  MoveL 6660 to (240.24, 47.55, 97.46) mm, rotated rx 180 ry 0 rz 180 deg; joints [-155.614, -72.061, -46.003, 43.936, 36.516, -37.754]
  Call Extruder(209.25610)
  MoveL 6661 to (240.29, 47.8, 97.46) mm, rotated rx 180 ry 0 rz 180 deg; joints [-155.594, -72.082, -45.96, 43.985, 36.511, -37.802]
  MoveL 6662 to (240.29, 47.8, 97.46) mm, rotated rx 180 ry 0 rz 180 deg; joints [-155.594, -72.082, -45.96, 43.985, 36.511, -37.802]
  Call Extruder(209.39246)
  MoveL 6663 to (240.34, 48.05, 97.46) mm, rotated rx -180 ry 0 rz 180 deg; joints [-155.574, -72.103, -45.916, 44.033, 36.507, -37.85]
  MoveL 6664 to (240.34, 48.05, 97.46) mm, rotated rx -180 ry 0 rz 180 deg; joints [-155.574, -72.103, -45.916, 44.033, 36.507, -37.85]
  Call Extruder(209.52822)
  MoveL 6665 to (240.39, 48.3, 97.46) mm, rotated rx -180 ry 0 rz 180 deg; joints [-155.554, -72.123, -45.873, 44.081, 36.503, -37.899]
  MoveL 6666 to (240.39, 48.3, 97.46) mm, rotated rx -180 ry 0 rz 180 deg; joints [-155.554, -72.123, -45.873, 44.081, 36.503, -37.899]
  Call Extruder(209.66337)
  MoveL 6667 to (240.44, 48.55, 97.46) mm, rotated rx 180 ry 0 rz 180 deg; joints [-155.534, -72.144, -45.829, 44.129, 36.499, -37.947]
  MoveL 6668 to (240.44, 48.55, 97.46) mm, rotated rx 180 ry 0 rz 180 deg; joints [-155.534, -72.144, -45.829, 44.129, 36.499, -37.947]
  Call Extruder(209.79791)
  MoveL 6669 to (240.49, 48.8, 97.46) mm, rotated rx 180 ry 0 rz 180 deg; joints [-155.514, -72.165, -45.785, 44.177, 36.495, -37.995]
  MoveL 6670 to (240.49, 48.8, 97.46) mm, rotated rx 180 ry 0 rz 180 deg; joints [-155.514, -72.165, -45.785, 44.177, 36.495, -37.995]
  Call Extruder(209.93183)
  MoveL 6671 to (240.54, 49.05, 97.46) mm, rotated rx 180 ry 0 rz -180 deg; joints [-155.494, -72.186, -45.742, 44.226, 36.491, -38.043]
  MoveL 6672 to (240.54, 49.05, 97.46) mm, rotated rx 180 ry 0 rz -180 deg; joints [-155.494, -72.186, -45.742, 44.226, 36.491, -38.043]
  Call Extruder(210.07970)
  MoveL 6673 to (240.59, 49.33, 97.46) mm, rotated rx 180 ry 0 rz 180 deg; joints [-155.471, -72.208, -45.695, 44.279, 36.487, -38.096]
  MoveL 6674 to (240.59, 49.33, 97.46) mm, rotated rx 180 ry 0 rz 180 deg; joints [-155.471, -72.208, -45.695, 44.279, 36.487, -38.096]
  Call Extruder(210.24144)
  MoveL 6675 to (240.64, 49.63, 97.46) mm, rotated rx 180 ry 0 rz -180 deg; joints [-155.446, -72.232, -45.644, 44.337, 36.484, -38.154]
  MoveL 6676 to (240.64, 49.63, 97.46) mm, rotated rx 180 ry 0 rz -180 deg; joints [-155.446, -72.232, -45.644, 44.337, 36.484, -38.154]
  Call Extruder(210.40246)
  MoveL 6677 to (240.69, 49.94, 97.46) mm, rotated rx 180 ry 0 rz 180 deg; joints [-155.421, -72.256, -45.593, 44.395, 36.481, -38.212]
  MoveL 6678 to (240.69, 49.94, 97.46) mm, rotated rx 180 ry 0 rz 180 deg; joints [-155.421, -72.256, -45.593, 44.395, 36.481, -38.212]
  Call Extruder(210.56275)
  MoveL 6679 to (240.74, 50.24, 97.46) mm, rotated rx -180 ry 0 rz 180 deg; joints [-155.396, -72.28, -45.543, 44.453, 36.477, -38.27]
  MoveL 6680 to (240.74, 50.24, 97.46) mm, rotated rx -180 ry 0 rz 180 deg; joints [-155.396, -72.28, -45.543, 44.453, 36.477, -38.27]
  Call Extruder(210.72231)
  MoveL 6681 to (240.78, 50.55, 97.46) mm, rotated rx 180 ry 0 rz 180 deg; joints [-155.371, -72.305, -45.492, 44.512, 36.474, -38.328]
  MoveL 6682 to (240.78, 50.55, 97.46) mm, rotated rx 180 ry 0 rz 180 deg; joints [-155.371, -72.305, -45.492, 44.512, 36.474, -38.328]
  Call Extruder(210.88114)
  MoveL 6683 to (240.83, 50.86, 97.46) mm, rotated rx -180 ry 0 rz 180 deg; joints [-155.346, -72.329, -45.441, 44.57, 36.47, -38.386]
  MoveL 6684 to (240.83, 50.86, 97.46) mm, rotated rx -180 ry 0 rz 180 deg; joints [-155.346, -72.329, -45.441, 44.57, 36.47, -38.386]
  Call Extruder(211.05982)
  MoveL 6685 to (240.88, 51.2, 97.46) mm, rotated rx -180 ry 0 rz 180 deg; joints [-155.317, -72.355, -45.386, 44.636, 36.467, -38.451]
  MoveL 6686 to (240.88, 51.2, 97.46) mm, rotated rx -180 ry 0 rz 180 deg; joints [-155.317, -72.355, -45.386, 44.636, 36.467, -38.451]
  Call Extruder(211.25826)
  MoveL 6687 to (240.93, 51.59, 97.46) mm, rotated rx 180 ry 0 rz -180 deg; joints [-155.285, -72.384, -45.325, 44.708, 36.465, -38.522]
  MoveL 6688 to (240.93, 51.59, 97.46) mm, rotated rx 180 ry 0 rz -180 deg; joints [-155.285, -72.384, -45.325, 44.708, 36.465, -38.522]
  Call Extruder(211.45583)
  MoveL 6689 to (240.97, 51.98, 97.46) mm, rotated rx 180 ry 0 rz 180 deg; joints [-155.252, -72.413, -45.264, 44.781, 36.463, -38.594]
  MoveL 6690 to (240.97, 51.98, 97.46) mm, rotated rx 180 ry 0 rz 180 deg; joints [-155.252, -72.413, -45.264, 44.781, 36.463, -38.594]
  Call Extruder(211.65254)
  MoveL 6691 to (241.02, 52.36, 97.46) mm, rotated rx 180 ry 0 rz 180 deg; joints [-155.22, -72.442, -45.204, 44.854, 36.46, -38.666]
  MoveL 6692 to (241.02, 52.36, 97.46) mm, rotated rx 180 ry 0 rz 180 deg; joints [-155.22, -72.442, -45.204, 44.854, 36.46, -38.666]
  Call Extruder(211.84838)
  MoveL 6693 to (241.06, 52.75, 97.46) mm, rotated rx 180 ry 0 rz 180 deg; joints [-155.188, -72.471, -45.143, 44.926, 36.458, -38.738]
  MoveL 6694 to (241.06, 52.75, 97.46) mm, rotated rx 180 ry 0 rz 180 deg; joints [-155.188, -72.471, -45.143, 44.926, 36.458, -38.738]
  Call Extruder(212.14382)
  MoveL 6695 to (241.11, 53.34, 97.46) mm, rotated rx 180 ry 0 rz 180 deg; joints [-155.138, -72.512, -45.057, 45.035, 36.457, -38.844]
  MoveL 6696 to (241.11, 53.34, 97.46) mm, rotated rx 180 ry 0 rz 180 deg; joints [-155.138, -72.512, -45.057, 45.035, 36.457, -38.844]
  Call Extruder(212.43792)
  MoveL 6697 to (241.16, 53.93, 97.46) mm, rotated rx 180 ry 0 rz 180 deg; joints [-155.088, -72.553, -44.97, 45.144, 36.457, -38.951]
  MoveL 6698 to (241.16, 53.93, 97.46) mm, rotated rx 180 ry 0 rz 180 deg; joints [-155.088, -72.553, -44.97, 45.144, 36.457, -38.951]
  Call Extruder(212.73070)
  MoveL 6699 to (241.2, 54.52, 97.46) mm, rotated rx 180 ry 0 rz -180 deg; joints [-155.038, -72.595, -44.883, 45.253, 36.456, -39.058]
  MoveL 6700 to (241.2, 54.52, 97.46) mm, rotated rx 180 ry 0 rz -180 deg; joints [-155.038, -72.595, -44.883, 45.253, 36.456, -39.058]
  Call Extruder(213.30415)
  MoveL 6701 to (241.25, 55.68, 97.46) mm, rotated rx 180 ry 0 rz 180 deg; joints [-154.938, -72.671, -44.724, 45.464, 36.461, -39.263]
  MoveL 6702 to (241.25, 55.68, 97.46) mm, rotated rx 180 ry 0 rz 180 deg; joints [-154.938, -72.671, -44.724, 45.464, 36.461, -39.263]
  Call Extruder(214.01798)
  MoveL 6703 to (241.29, 57.14, 97.46) mm, rotated rx 180 ry 0 rz -180 deg; joints [-154.812, -72.765, -44.527, 45.727, 36.469, -39.518]
  Call Extruder(256.08287)
  MoveL 6704 to (241.29, 142.86, 97.46) mm, rotated rx 180 ry 0 rz 180 deg; joints [-147.778, -79.586, -30.484, 61.433, 37.381, -55.581]
  Call Extruder(256.51129)
  MoveL 6705 to (241.27, 143.73, 97.46) mm, rotated rx 180 ry 0 rz 180 deg; joints [-147.711, -79.673, -30.306, 61.599, 37.394, -55.761]
  MoveL 6706 to (241.27, 143.73, 97.46) mm, rotated rx 180 ry 0 rz 180 deg; joints [-147.711, -79.673, -30.306, 61.599, 37.394, -55.761]
  Call Extruder(257.08474)
  MoveL 6707 to (241.22, 144.9, 97.46) mm, rotated rx -180 ry 0 rz -180 deg; joints [-147.62, -79.787, -30.075, 61.818, 37.413, -55.998]
  MoveL 6708 to (241.22, 144.9, 97.46) mm, rotated rx -180 ry 0 rz -180 deg; joints [-147.62, -79.787, -30.075, 61.818, 37.413, -55.998]
  Call Extruder(257.51908)
  MoveL 6709 to (241.18, 145.77, 97.46) mm, rotated rx 180 ry 0 rz 180 deg; joints [-147.551, -79.872, -29.904, 61.981, 37.43, -56.174]
  MoveL 6710 to (241.18, 145.77, 97.46) mm, rotated rx 180 ry 0 rz 180 deg; joints [-147.551, -79.872, -29.904, 61.981, 37.43, -56.174]
  Call Extruder(257.81319)
  MoveL 6711 to (241.13, 146.36, 97.46) mm, rotated rx -180 ry 0 rz -180 deg; joints [-147.504, -79.926, -29.794, 62.089, 37.443, -56.289]
  MoveL 6712 to (241.13, 146.36, 97.46) mm, rotated rx -180 ry 0 rz -180 deg; joints [-147.504, -79.926, -29.794, 62.089, 37.443, -56.289]
  Call Extruder(258.10863)
  MoveL 6713 to (241.09, 146.95, 97.46) mm, rotated rx -180 ry 0 rz 180 deg; joints [-147.457, -79.981, -29.682, 62.197, 37.456, -56.405]
  MoveL 6714 to (241.09, 146.95, 97.46) mm, rotated rx -180 ry 0 rz 180 deg; joints [-147.457, -79.981, -29.682, 62.197, 37.456, -56.405]
  Call Extruder(258.35489)
  MoveL 6715 to (241.04, 147.44, 97.46) mm, rotated rx 180 ry 0 rz 180 deg; joints [-147.417, -80.026, -29.593, 62.285, 37.467, -56.499]
  MoveL 6716 to (241.04, 147.44, 97.46) mm, rotated rx 180 ry 0 rz 180 deg; joints [-147.417, -80.026, -29.593, 62.285, 37.467, -56.499]
  Call Extruder(258.55159)
  MoveL 6717 to (240.99, 147.83, 97.46) mm, rotated rx 180 ry 0 rz 180 deg; joints [-147.386, -80.059, -29.524, 62.353, 37.478, -56.572]
  MoveL 6718 to (240.99, 147.83, 97.46) mm, rotated rx 180 ry 0 rz 180 deg; joints [-147.386, -80.059, -29.524, 62.353, 37.478, -56.572]
  Call Extruder(258.74917)
  MoveL 6719 to (240.95, 148.22, 97.46) mm, rotated rx 180 ry 0 rz 180 deg; joints [-147.354, -80.093, -29.456, 62.422, 37.488, -56.645]
  MoveL 6720 to (240.95, 148.22, 97.46) mm, rotated rx 180 ry 0 rz 180 deg; joints [-147.354, -80.093, -29.456, 62.422, 37.488, -56.645]
  Call Extruder(258.94761)
  MoveL 6721 to (240.9, 148.6, 97.46) mm, rotated rx -180 ry 0 rz -180 deg; joints [-147.322, -80.127, -29.387, 62.49, 37.499, -56.719]
  MoveL 6722 to (240.9, 148.6, 97.46) mm, rotated rx -180 ry 0 rz -180 deg; joints [-147.322, -80.127, -29.387, 62.49, 37.499, -56.719]
  Call Extruder(259.14692)
  MoveL 6723 to (240.86, 148.99, 97.46) mm, rotated rx -180 ry 0 rz 180 deg; joints [-147.291, -80.161, -29.319, 62.559, 37.509, -56.792]
  MoveL 6724 to (240.86, 148.99, 97.46) mm, rotated rx -180 ry 0 rz 180 deg; joints [-147.291, -80.161, -29.319, 62.559, 37.509, -56.792]
  Call Extruder(259.30575)
  MoveL 6725 to (240.81, 149.3, 97.46) mm, rotated rx 180 ry 0 rz 180 deg; joints [-147.265, -80.186, -29.268, 62.611, 37.518, -56.847]
  MoveL 6726 to (240.81, 149.3, 97.46) mm, rotated rx 180 ry 0 rz 180 deg; joints [-147.265, -80.186, -29.268, 62.611, 37.518, -56.847]
  Call Extruder(259.46531)
  MoveL 6727 to (240.76, 149.6, 97.46) mm, rotated rx -180 ry 0 rz -180 deg; joints [-147.24, -80.211, -29.218, 62.664, 37.528, -56.902]
  MoveL 6728 to (240.76, 149.6, 97.46) mm, rotated rx -180 ry 0 rz -180 deg; joints [-147.24, -80.211, -29.218, 62.664, 37.528, -56.902]
  Call Extruder(259.62559)
  MoveL 6729 to (240.71, 149.91, 97.46) mm, rotated rx 180 ry 0 rz 180 deg; joints [-147.214, -80.236, -29.168, 62.716, 37.538, -56.958]
  MoveL 6730 to (240.71, 149.91, 97.46) mm, rotated rx 180 ry 0 rz 180 deg; joints [-147.214, -80.236, -29.168, 62.716, 37.538, -56.958]
  Call Extruder(259.78661)
  MoveL 6731 to (240.66, 150.21, 97.46) mm, rotated rx 180 ry 0 rz 180 deg; joints [-147.189, -80.261, -29.117, 62.768, 37.548, -57.013]
  MoveL 6732 to (240.66, 150.21, 97.46) mm, rotated rx 180 ry 0 rz 180 deg; joints [-147.189, -80.261, -29.117, 62.768, 37.548, -57.013]
  Call Extruder(259.94835)
  MoveL 6733 to (240.61, 150.52, 97.46) mm, rotated rx 180 ry 0 rz 180 deg; joints [-147.163, -80.286, -29.066, 62.821, 37.557, -57.068]
  MoveL 6734 to (240.61, 150.52, 97.46) mm, rotated rx 180 ry 0 rz 180 deg; joints [-147.163, -80.286, -29.066, 62.821, 37.557, -57.068]
  Call Extruder(260.11082)
  MoveL 6735 to (240.56, 150.83, 97.46) mm, rotated rx 180 ry 0 rz -180 deg; joints [-147.138, -80.311, -29.016, 62.873, 37.567, -57.124]
  MoveL 6736 to (240.56, 150.83, 97.46) mm, rotated rx 180 ry 0 rz -180 deg; joints [-147.138, -80.311, -29.016, 62.873, 37.567, -57.124]
  Call Extruder(260.24475)
  MoveL 6737 to (240.52, 151.07, 97.46) mm, rotated rx 180 ry 0 rz 180 deg; joints [-147.117, -80.33, -28.977, 62.914, 37.576, -57.167]
  MoveL 6738 to (240.52, 151.07, 97.46) mm, rotated rx 180 ry 0 rz 180 deg; joints [-147.117, -80.33, -28.977, 62.914, 37.576, -57.167]
  Call Extruder(260.37929)
  MoveL 6739 to (240.47, 151.32, 97.46) mm, rotated rx -180 ry 0 rz 180 deg; joints [-147.095, -80.349, -28.939, 62.955, 37.585, -57.21]
  MoveL 6740 to (240.47, 151.32, 97.46) mm, rotated rx -180 ry 0 rz 180 deg; joints [-147.095, -80.349, -28.939, 62.955, 37.585, -57.21]
  Call Extruder(260.51443)
  MoveL 6741 to (240.42, 151.57, 97.46) mm, rotated rx 180 ry 0 rz 180 deg; joints [-147.074, -80.368, -28.901, 62.996, 37.594, -57.253]
  MoveL 6742 to (240.42, 151.57, 97.46) mm, rotated rx 180 ry 0 rz 180 deg; joints [-147.074, -80.368, -28.901, 62.996, 37.594, -57.253]
  Call Extruder(260.65019)
  MoveL 6743 to (240.37, 151.82, 97.46) mm, rotated rx 180 ry 0 rz -180 deg; joints [-147.053, -80.387, -28.863, 63.038, 37.603, -57.296]
  MoveL 6744 to (240.37, 151.82, 97.46) mm, rotated rx 180 ry 0 rz -180 deg; joints [-147.053, -80.387, -28.863, 63.038, 37.603, -57.296]
  Call Extruder(260.78656)
  MoveL 6745 to (240.32, 152.07, 97.46) mm, rotated rx 180 ry 0 rz 180 deg; joints [-147.032, -80.406, -28.825, 63.079, 37.612, -57.339]
  MoveL 6746 to (240.32, 152.07, 97.46) mm, rotated rx 180 ry 0 rz 180 deg; joints [-147.032, -80.406, -28.825, 63.079, 37.612, -57.339]
  Call Extruder(260.92354)
  MoveL 6747 to (240.27, 152.32, 97.46) mm, rotated rx 180 ry 0 rz 180 deg; joints [-147.011, -80.425, -28.786, 63.12, 37.621, -57.382]
  MoveL 6748 to (240.27, 152.32, 97.46) mm, rotated rx 180 ry 0 rz 180 deg; joints [-147.011, -80.425, -28.786, 63.12, 37.621, -57.382]
  Call Extruder(261.06113)
  MoveL 6749 to (240.22, 152.57, 97.46) mm, rotated rx 180 ry 0 rz 180 deg; joints [-146.989, -80.444, -28.748, 63.161, 37.63, -57.425]
  MoveL 6750 to (240.22, 152.57, 97.46) mm, rotated rx 180 ry 0 rz 180 deg; joints [-146.989, -80.444, -28.748, 63.161, 37.63, -57.425]
  Call Extruder(261.17482)
  MoveL 6751 to (240.17, 152.77, 97.46) mm, rotated rx 180 ry 0 rz 180 deg; joints [-146.972, -80.459, -28.717, 63.194, 37.638, -57.46]
  MoveL 6752 to (240.17, 152.77, 97.46) mm, rotated rx 180 ry 0 rz 180 deg; joints [-146.972, -80.459, -28.717, 63.194, 37.638, -57.46]
  Call Extruder(261.28897)
  MoveL 6753 to (240.13, 152.98, 97.46) mm, rotated rx -180 ry 0 rz -180 deg; joints [-146.954, -80.474, -28.687, 63.228, 37.646, -57.495]
  MoveL 6754 to (240.13, 152.98, 97.46) mm, rotated rx -180 ry 0 rz -180 deg; joints [-146.954, -80.474, -28.687, 63.228, 37.646, -57.495]
  Call Extruder(261.40358)
  MoveL 6755 to (240.08, 153.18, 97.46) mm, rotated rx -180 ry 0 rz 180 deg; joints [-146.937, -80.489, -28.657, 63.261, 37.654, -57.529]
  MoveL 6756 to (240.08, 153.18, 97.46) mm, rotated rx -180 ry 0 rz 180 deg; joints [-146.937, -80.489, -28.657, 63.261, 37.654, -57.529]
  Call Extruder(261.51863)
  MoveL 6757 to (240.04, 153.39, 97.46) mm, rotated rx 180 ry 0 rz -180 deg; joints [-146.919, -80.504, -28.627, 63.294, 37.662, -57.564]
  MoveL 6758 to (240.04, 153.39, 97.46) mm, rotated rx 180 ry 0 rz -180 deg; joints [-146.919, -80.504, -28.627, 63.294, 37.662, -57.564]
  Call Extruder(261.64086)
  MoveL 6759 to (239.98, 153.6, 97.46) mm, rotated rx -180 ry 0 rz 180 deg; joints [-146.9, -80.518, -28.598, 63.327, 37.671, -57.598]
  MoveL 6760 to (239.98, 153.6, 97.46) mm, rotated rx -180 ry 0 rz 180 deg; joints [-146.9, -80.518, -28.598, 63.327, 37.671, -57.598]
  Call Extruder(261.77052)
  MoveL 6761 to (239.92, 153.82, 97.46) mm, rotated rx -180 ry 0 rz 180 deg; joints [-146.88, -80.531, -28.571, 63.36, 37.682, -57.632]
  MoveL 6762 to (239.92, 153.82, 97.46) mm, rotated rx -180 ry 0 rz 180 deg; joints [-146.88, -80.531, -28.571, 63.36, 37.682, -57.632]
  Call Extruder(261.90074)
  MoveL 6763 to (239.85, 154.05, 97.46) mm, rotated rx 180 ry 0 rz 180 deg; joints [-146.86, -80.544, -28.544, 63.394, 37.693, -57.665]
  MoveL 6764 to (239.85, 154.05, 97.46) mm, rotated rx 180 ry 0 rz 180 deg; joints [-146.86, -80.544, -28.544, 63.394, 37.693, -57.665]
  Call Extruder(262.03153)
  MoveL 6765 to (239.78, 154.27, 97.46) mm, rotated rx 180 ry 0 rz -180 deg; joints [-146.84, -80.558, -28.517, 63.427, 37.704, -57.7]
  MoveL 6766 to (239.78, 154.27, 97.46) mm, rotated rx 180 ry 0 rz -180 deg; joints [-146.84, -80.558, -28.517, 63.427, 37.704, -57.7]
  Call Extruder(262.16289)
  MoveL 6767 to (239.71, 154.49, 97.46) mm, rotated rx -180 ry 0 rz 180 deg; joints [-146.82, -80.571, -28.49, 63.46, 37.715, -57.733]
  MoveL 6768 to (239.71, 154.49, 97.46) mm, rotated rx -180 ry 0 rz 180 deg; joints [-146.82, -80.571, -28.49, 63.46, 37.715, -57.733]
  Call Extruder(262.27479)
  MoveL 6769 to (239.65, 154.68, 97.46) mm, rotated rx -180 ry 0 rz 180 deg; joints [-146.803, -80.582, -28.469, 63.488, 37.725, -57.761]
  MoveL 6770 to (239.65, 154.68, 97.46) mm, rotated rx -180 ry 0 rz 180 deg; joints [-146.803, -80.582, -28.469, 63.488, 37.725, -57.761]
  Call Extruder(262.38714)
  MoveL 6771 to (239.59, 154.87, 97.46) mm, rotated rx 180 ry 0 rz 180 deg; joints [-146.785, -80.592, -28.447, 63.515, 37.735, -57.789]
  MoveL 6772 to (239.59, 154.87, 97.46) mm, rotated rx 180 ry 0 rz 180 deg; joints [-146.785, -80.592, -28.447, 63.515, 37.735, -57.789]
  Call Extruder(262.49993)
  MoveL 6773 to (239.53, 155.06, 97.46) mm, rotated rx 180 ry 0 rz -180 deg; joints [-146.768, -80.603, -28.426, 63.543, 37.744, -57.816]
  MoveL 6774 to (239.53, 155.06, 97.46) mm, rotated rx 180 ry 0 rz -180 deg; joints [-146.768, -80.603, -28.426, 63.543, 37.744, -57.816]
  Call Extruder(262.61316)
  MoveL 6775 to (239.47, 155.25, 97.46) mm, rotated rx 180 ry 0 rz -180 deg; joints [-146.751, -80.614, -28.405, 63.57, 37.754, -57.844]
  MoveL 6776 to (239.47, 155.25, 97.46) mm, rotated rx 180 ry 0 rz -180 deg; joints [-146.751, -80.614, -28.405, 63.57, 37.754, -57.844]
  Call Extruder(262.72684)
  MoveL 6777 to (239.41, 155.44, 97.46) mm, rotated rx -180 ry 0 rz 180 deg; joints [-146.734, -80.624, -28.383, 63.598, 37.764, -57.871]
  MoveL 6778 to (239.41, 155.44, 97.46) mm, rotated rx -180 ry 0 rz 180 deg; joints [-146.734, -80.624, -28.383, 63.598, 37.764, -57.871]
  Call Extruder(262.90880)
  MoveL 6779 to (239.29, 155.73, 97.46) mm, rotated rx 180 ry 0 rz 180 deg; joints [-146.706, -80.636, -28.359, 63.636, 37.782, -57.909]
  MoveL 6780 to (239.29, 155.73, 97.46) mm, rotated rx 180 ry 0 rz 180 deg; joints [-146.706, -80.636, -28.359, 63.636, 37.782, -57.909]
  Call Extruder(263.09151)
  MoveL 6781 to (239.17, 156.02, 97.46) mm, rotated rx 180 ry 0 rz -180 deg; joints [-146.678, -80.648, -28.334, 63.674, 37.8, -57.946]
  MoveL 6782 to (239.17, 156.02, 97.46) mm, rotated rx 180 ry 0 rz -180 deg; joints [-146.678, -80.648, -28.334, 63.674, 37.8, -57.946]
  Call Extruder(263.26194)
  MoveL 6783 to (239.05, 156.29, 97.46) mm, rotated rx -180 ry 0 rz -180 deg; joints [-146.652, -80.659, -28.312, 63.71, 37.817, -57.98]
  MoveL 6784 to (239.05, 156.29, 97.46) mm, rotated rx -180 ry 0 rz -180 deg; joints [-146.652, -80.659, -28.312, 63.71, 37.817, -57.98]
  Call Extruder(263.41995)
  MoveL 6785 to (238.94, 156.54, 97.46) mm, rotated rx 180 ry 0 rz 180 deg; joints [-146.628, -80.669, -28.293, 63.742, 37.833, -58.01]
  MoveL 6786 to (238.94, 156.54, 97.46) mm, rotated rx 180 ry 0 rz 180 deg; joints [-146.628, -80.669, -28.293, 63.742, 37.833, -58.01]
  Call Extruder(263.57856)
  MoveL 6787 to (238.84, 156.79, 97.46) mm, rotated rx 180 ry 0 rz 180 deg; joints [-146.604, -80.679, -28.273, 63.774, 37.849, -58.041]
  MoveL 6788 to (238.84, 156.79, 97.46) mm, rotated rx 180 ry 0 rz 180 deg; joints [-146.604, -80.679, -28.273, 63.774, 37.849, -58.041]
  Call Extruder(263.78473)
  MoveL 6789 to (238.66, 157.09, 97.46) mm, rotated rx -180 ry 0 rz 180 deg; joints [-146.573, -80.683, -28.264, 63.806, 37.873, -58.069]
  MoveL 6790 to (238.66, 157.09, 97.46) mm, rotated rx -180 ry 0 rz 180 deg; joints [-146.573, -80.683, -28.264, 63.806, 37.873, -58.069]
  Call Extruder(263.99168)
  MoveL 6791 to (238.49, 157.4, 97.46) mm, rotated rx -180 ry 0 rz 180 deg; joints [-146.542, -80.688, -28.255, 63.838, 37.898, -58.097]
  MoveL 6792 to (238.49, 157.4, 97.46) mm, rotated rx -180 ry 0 rz 180 deg; joints [-146.542, -80.688, -28.255, 63.838, 37.898, -58.097]
  Call Extruder(264.19941)
  MoveL 6793 to (238.31, 157.7, 97.46) mm, rotated rx 180 ry 0 rz -180 deg; joints [-146.51, -80.692, -28.246, 63.87, 37.923, -58.125]
  MoveL 6794 to (238.31, 157.7, 97.46) mm, rotated rx 180 ry 0 rz -180 deg; joints [-146.51, -80.692, -28.246, 63.87, 37.923, -58.125]
  Call Extruder(264.40791)
  MoveL 6795 to (238.14, 158.01, 97.46) mm, rotated rx -180 ry 0 rz 180 deg; joints [-146.479, -80.696, -28.238, 63.902, 37.948, -58.153]
  MoveL 6796 to (238.14, 158.01, 97.46) mm, rotated rx -180 ry 0 rz 180 deg; joints [-146.479, -80.696, -28.238, 63.902, 37.948, -58.153]
  Call Extruder(264.58745)
  MoveL 6797 to (237.96, 158.25, 97.46) mm, rotated rx 180 ry 0 rz -180 deg; joints [-146.452, -80.694, -28.242, 63.923, 37.972, -58.167]
  MoveL 6798 to (237.96, 158.25, 97.46) mm, rotated rx 180 ry 0 rz -180 deg; joints [-146.452, -80.694, -28.242, 63.923, 37.972, -58.167]
  Call Extruder(264.92086)
  MoveL 6799 to (237.63, 158.7, 97.46) mm, rotated rx 180 ry 0 rz -180 deg; joints [-146.402, -80.689, -28.252, 63.96, 38.016, -58.194]
  MoveL 6800 to (237.63, 158.7, 97.46) mm, rotated rx 180 ry 0 rz -180 deg; joints [-146.402, -80.689, -28.252, 63.96, 38.016, -58.194]
  Call Extruder(265.25545)
  MoveL 6801 to (237.3, 159.15, 97.46) mm, rotated rx -180 ry 0 rz 180 deg; joints [-146.352, -80.684, -28.262, 63.997, 38.061, -58.221]
  Call Extruder(266.08341)
  MoveL 6802 to (236.39, 160.19, 97.46) mm, rotated rx -180 ry 0 rz 180 deg; joints [-146.229, -80.647, -28.337, 64.058, 38.182, -58.247]
  Call Extruder(266.91134)
  MoveL 6803 to (235.35, 161.1, 97.46) mm, rotated rx 180 ry 0 rz 180 deg; joints [-146.109, -80.575, -28.483, 64.076, 38.316, -58.22]
  Call Extruder(267.07865)
  MoveL 6804 to (235.13, 161.27, 97.46) mm, rotated rx -180 ry 0 rz 180 deg; joints [-146.086, -80.555, -28.523, 64.073, 38.345, -58.207]
  MoveL 6805 to (235.13, 161.27, 97.46) mm, rotated rx -180 ry 0 rz 180 deg; joints [-146.086, -80.555, -28.523, 64.073, 38.345, -58.207]
  Call Extruder(267.41207)
  MoveL 6806 to (234.68, 161.59, 97.46) mm, rotated rx 180 ry 0 rz 180 deg; joints [-146.039, -80.516, -28.601, 64.068, 38.402, -58.181]
  MoveL 6807 to (234.68, 161.59, 97.46) mm, rotated rx 180 ry 0 rz 180 deg; joints [-146.039, -80.516, -28.601, 64.068, 38.402, -58.181]
  Call Extruder(267.74432)
  MoveL 6808 to (234.22, 161.92, 97.46) mm, rotated rx 180 ry 0 rz 180 deg; joints [-145.992, -80.478, -28.679, 64.064, 38.459, -58.155]
  MoveL 6809 to (234.22, 161.92, 97.46) mm, rotated rx 180 ry 0 rz 180 deg; joints [-145.992, -80.478, -28.679, 64.064, 38.459, -58.155]
  Call Extruder(267.86197)
  MoveL 6810 to (234.05, 162.02, 97.46) mm, rotated rx 180 ry 0 rz 180 deg; joints [-145.976, -80.46, -28.715, 64.057, 38.481, -58.14]
  MoveL 6811 to (234.05, 162.02, 97.46) mm, rotated rx 180 ry 0 rz 180 deg; joints [-145.976, -80.46, -28.715, 64.057, 38.481, -58.14]
  Call Extruder(268.06970)
  MoveL 6812 to (233.75, 162.2, 97.46) mm, rotated rx -180 ry 0 rz 180 deg; joints [-145.947, -80.429, -28.777, 64.045, 38.519, -58.113]
  MoveL 6813 to (233.75, 162.2, 97.46) mm, rotated rx -180 ry 0 rz 180 deg; joints [-145.947, -80.429, -28.777, 64.045, 38.519, -58.113]
  Call Extruder(268.27665)
  MoveL 6814 to (233.45, 162.37, 97.46) mm, rotated rx 180 ry 0 rz 180 deg; joints [-145.919, -80.398, -28.84, 64.034, 38.557, -58.086]
  MoveL 6815 to (233.45, 162.37, 97.46) mm, rotated rx 180 ry 0 rz 180 deg; joints [-145.919, -80.398, -28.84, 64.034, 38.557, -58.086]
  Call Extruder(268.48282)
  MoveL 6816 to (233.14, 162.55, 97.46) mm, rotated rx 180 ry 0 rz -180 deg; joints [-145.891, -80.367, -28.903, 64.022, 38.594, -58.059]
  MoveL 6817 to (233.14, 162.55, 97.46) mm, rotated rx 180 ry 0 rz -180 deg; joints [-145.891, -80.367, -28.903, 64.022, 38.594, -58.059]
  Call Extruder(268.66449)
  MoveL 6818 to (232.87, 162.69, 97.46) mm, rotated rx -180 ry 0 rz 180 deg; joints [-145.866, -80.337, -28.964, 64.008, 38.629, -58.031]
  MoveL 6819 to (232.87, 162.69, 97.46) mm, rotated rx -180 ry 0 rz 180 deg; joints [-145.866, -80.337, -28.964, 64.008, 38.629, -58.031]
  Call Extruder(268.82246)
  MoveL 6820 to (232.62, 162.8, 97.46) mm, rotated rx 180 ry 0 rz 180 deg; joints [-145.845, -80.307, -29.023, 63.992, 38.659, -58.002]
  MoveL 6821 to (232.62, 162.8, 97.46) mm, rotated rx 180 ry 0 rz 180 deg; joints [-145.845, -80.307, -29.023, 63.992, 38.659, -58.002]
  Call Extruder(268.97983)
  MoveL 6822 to (232.37, 162.9, 97.46) mm, rotated rx 180 ry 0 rz 180 deg; joints [-145.825, -80.278, -29.082, 63.976, 38.69, -57.972]
  MoveL 6823 to (232.37, 162.9, 97.46) mm, rotated rx 180 ry 0 rz 180 deg; joints [-145.825, -80.278, -29.082, 63.976, 38.69, -57.972]
  Call Extruder(269.16257)
  MoveL 6824 to (232.07, 163.02, 97.46) mm, rotated rx 180 ry 0 rz 180 deg; joints [-145.801, -80.243, -29.153, 63.956, 38.726, -57.937]
  MoveL 6825 to (232.07, 163.02, 97.46) mm, rotated rx 180 ry 0 rz 180 deg; joints [-145.801, -80.243, -29.153, 63.956, 38.726, -57.937]
  Call Extruder(269.34456)
  MoveL 6826 to (231.78, 163.15, 97.46) mm, rotated rx 180 ry 0 rz 180 deg; joints [-145.777, -80.208, -29.223, 63.936, 38.761, -57.902]
  MoveL 6827 to (231.78, 163.15, 97.46) mm, rotated rx 180 ry 0 rz 180 deg; joints [-145.777, -80.208, -29.223, 63.936, 38.761, -57.902]
  Call Extruder(269.49190)
  MoveL 6828 to (231.54, 163.24, 97.46) mm, rotated rx 180 ry 0 rz 180 deg; joints [-145.759, -80.179, -29.283, 63.919, 38.791, -57.871]
  MoveL 6829 to (231.54, 163.24, 97.46) mm, rotated rx 180 ry 0 rz 180 deg; joints [-145.759, -80.179, -29.283, 63.919, 38.791, -57.871]
  Call Extruder(269.60512)
  MoveL 6830 to (231.35, 163.3, 97.46) mm, rotated rx 180 ry 0 rz 180 deg; joints [-145.744, -80.155, -29.332, 63.903, 38.813, -57.845]
  MoveL 6831 to (231.35, 163.3, 97.46) mm, rotated rx 180 ry 0 rz 180 deg; joints [-145.744, -80.155, -29.332, 63.903, 38.813, -57.845]
  Call Extruder(269.71789)
  MoveL 6832 to (231.17, 163.36, 97.46) mm, rotated rx 180 ry 0 rz 180 deg; joints [-145.73, -80.131, -29.38, 63.887, 38.836, -57.819]
  MoveL 6833 to (231.17, 163.36, 97.46) mm, rotated rx 180 ry 0 rz 180 deg; joints [-145.73, -80.131, -29.38, 63.887, 38.836, -57.819]
  Call Extruder(269.83022)
  MoveL 6834 to (230.98, 163.42, 97.46) mm, rotated rx 180 ry 0 rz 180 deg; joints [-145.716, -80.106, -29.429, 63.872, 38.859, -57.793]
  MoveL 6835 to (230.98, 163.42, 97.46) mm, rotated rx 180 ry 0 rz 180 deg; joints [-145.716, -80.106, -29.429, 63.872, 38.859, -57.793]
  Call Extruder(269.94211)
  MoveL 6836 to (230.79, 163.48, 97.46) mm, rotated rx -180 ry 0 rz -180 deg; joints [-145.702, -80.082, -29.478, 63.856, 38.882, -57.767]
  MoveL 6837 to (230.79, 163.48, 97.46) mm, rotated rx -180 ry 0 rz -180 deg; joints [-145.702, -80.082, -29.478, 63.856, 38.882, -57.767]
  Call Extruder(270.06351)
  MoveL 6838 to (230.58, 163.55, 97.46) mm, rotated rx 180 ry 0 rz 180 deg; joints [-145.687, -80.056, -29.532, 63.839, 38.907, -57.738]
  MoveL 6839 to (230.58, 163.55, 97.46) mm, rotated rx 180 ry 0 rz 180 deg; joints [-145.687, -80.056, -29.532, 63.839, 38.907, -57.738]
  Call Extruder(270.19433)
  MoveL 6840 to (230.36, 163.61, 97.46) mm, rotated rx 180 ry 0 rz 180 deg; joints [-145.67, -80.027, -29.591, 63.82, 38.934, -57.707]
  MoveL 6841 to (230.36, 163.61, 97.46) mm, rotated rx 180 ry 0 rz 180 deg; joints [-145.67, -80.027, -29.591, 63.82, 38.934, -57.707]
  Call Extruder(270.32458)
  MoveL 6842 to (230.14, 163.68, 97.46) mm, rotated rx 180 ry 0 rz 180 deg; joints [-145.654, -79.998, -29.649, 63.801, 38.961, -57.675]
  MoveL 6843 to (230.14, 163.68, 97.46) mm, rotated rx 180 ry 0 rz 180 deg; joints [-145.654, -79.998, -29.649, 63.801, 38.961, -57.675]
  Call Extruder(270.45426)
  MoveL 6844 to (229.91, 163.75, 97.46) mm, rotated rx -180 ry 0 rz 180 deg; joints [-145.638, -79.969, -29.708, 63.782, 38.988, -57.644]
  MoveL 6845 to (229.91, 163.75, 97.46) mm, rotated rx -180 ry 0 rz 180 deg; joints [-145.638, -79.969, -29.708, 63.782, 38.988, -57.644]
  Call Extruder(270.58338)
  MoveL 6846 to (229.69, 163.82, 97.46) mm, rotated rx 180 ry 0 rz 180 deg; joints [-145.621, -79.94, -29.767, 63.763, 39.015, -57.612]
  MoveL 6847 to (229.69, 163.82, 97.46) mm, rotated rx 180 ry 0 rz 180 deg; joints [-145.621, -79.94, -29.767, 63.763, 39.015, -57.612]
  Call Extruder(270.69845)
  MoveL 6848 to (229.48, 163.86, 97.46) mm, rotated rx 180 ry 0 rz 180 deg; joints [-145.607, -79.912, -29.824, 63.743, 39.039, -57.58]
  MoveL 6849 to (229.48, 163.86, 97.46) mm, rotated rx 180 ry 0 rz 180 deg; joints [-145.607, -79.912, -29.824, 63.743, 39.039, -57.58]
  Call Extruder(270.81308)
  MoveL 6850 to (229.28, 163.91, 97.46) mm, rotated rx 180 ry 0 rz -180 deg; joints [-145.594, -79.883, -29.881, 63.723, 39.063, -57.548]
  MoveL 6851 to (229.28, 163.91, 97.46) mm, rotated rx 180 ry 0 rz -180 deg; joints [-145.594, -79.883, -29.881, 63.723, 39.063, -57.548]
  Call Extruder(270.92725)
  MoveL 6852 to (229.08, 163.95, 97.46) mm, rotated rx 180 ry 0 rz -180 deg; joints [-145.58, -79.855, -29.938, 63.702, 39.088, -57.516]
  MoveL 6853 to (229.08, 163.95, 97.46) mm, rotated rx 180 ry 0 rz -180 deg; joints [-145.58, -79.855, -29.938, 63.702, 39.088, -57.516]
  Call Extruder(271.04096)
  MoveL 6854 to (228.87, 164, 97.46) mm, rotated rx 180 ry 0 rz 180 deg; joints [-145.566, -79.827, -29.995, 63.682, 39.112, -57.484]
  MoveL 6855 to (228.87, 164, 97.46) mm, rotated rx 180 ry 0 rz 180 deg; joints [-145.566, -79.827, -29.995, 63.682, 39.112, -57.484]
  Call Extruder(271.16638)
  MoveL 6856 to (228.65, 164.04, 97.46) mm, rotated rx 180 ry 0 rz 180 deg; joints [-145.551, -79.796, -30.058, 63.66, 39.139, -57.448]
  MoveL 6857 to (228.65, 164.04, 97.46) mm, rotated rx 180 ry 0 rz 180 deg; joints [-145.551, -79.796, -30.058, 63.66, 39.139, -57.448]
  Call Extruder(271.30336)
  MoveL 6858 to (228.4, 164.09, 97.46) mm, rotated rx 180 ry 0 rz 180 deg; joints [-145.535, -79.761, -30.128, 63.635, 39.169, -57.409]
  MoveL 6859 to (228.4, 164.09, 97.46) mm, rotated rx 180 ry 0 rz 180 deg; joints [-145.535, -79.761, -30.128, 63.635, 39.169, -57.409]
  Call Extruder(271.43973)
  MoveL 6860 to (228.15, 164.14, 97.46) mm, rotated rx -180 ry 0 rz 180 deg; joints [-145.518, -79.726, -30.199, 63.609, 39.198, -57.369]
  MoveL 6861 to (228.15, 164.14, 97.46) mm, rotated rx -180 ry 0 rz 180 deg; joints [-145.518, -79.726, -30.199, 63.609, 39.198, -57.369]
  Call Extruder(271.57549)
  MoveL 6862 to (227.9, 164.19, 97.46) mm, rotated rx 180 ry 0 rz 180 deg; joints [-145.502, -79.692, -30.269, 63.585, 39.228, -57.33]
  MoveL 6863 to (227.9, 164.19, 97.46) mm, rotated rx 180 ry 0 rz 180 deg; joints [-145.502, -79.692, -30.269, 63.585, 39.228, -57.33]
  Call Extruder(271.71064)
  MoveL 6864 to (227.65, 164.24, 97.46) mm, rotated rx 180 ry 0 rz 180 deg; joints [-145.485, -79.657, -30.339, 63.56, 39.258, -57.29]
  MoveL 6865 to (227.65, 164.24, 97.46) mm, rotated rx 180 ry 0 rz 180 deg; joints [-145.485, -79.657, -30.339, 63.56, 39.258, -57.29]
  Call Extruder(271.84517)
  MoveL 6866 to (227.4, 164.29, 97.46) mm, rotated rx 180 ry 0 rz 180 deg; joints [-145.469, -79.623, -30.409, 63.535, 39.287, -57.251]
  MoveL 6867 to (227.4, 164.29, 97.46) mm, rotated rx 180 ry 0 rz 180 deg; joints [-145.469, -79.623, -30.409, 63.535, 39.287, -57.251]
  Call Extruder(271.97910)
  MoveL 6868 to (227.15, 164.34, 97.46) mm, rotated rx -180 ry 0 rz -180 deg; joints [-145.453, -79.588, -30.478, 63.511, 39.317, -57.212]
  MoveL 6869 to (227.15, 164.34, 97.46) mm, rotated rx -180 ry 0 rz -180 deg; joints [-145.453, -79.588, -30.478, 63.511, 39.317, -57.212]
  Call Extruder(272.12696)
  MoveL 6870 to (226.87, 164.39, 97.46) mm, rotated rx 180 ry 0 rz -180 deg; joints [-145.435, -79.55, -30.557, 63.482, 39.35, -57.168]
  MoveL 6871 to (226.87, 164.39, 97.46) mm, rotated rx 180 ry 0 rz -180 deg; joints [-145.435, -79.55, -30.557, 63.482, 39.35, -57.168]
  Call Extruder(272.28870)
  MoveL 6872 to (226.57, 164.44, 97.46) mm, rotated rx 180 ry 0 rz -180 deg; joints [-145.415, -79.506, -30.645, 63.45, 39.386, -57.118]
  MoveL 6873 to (226.57, 164.44, 97.46) mm, rotated rx 180 ry 0 rz -180 deg; joints [-145.415, -79.506, -30.645, 63.45, 39.386, -57.118]
  Call Extruder(272.44972)
  MoveL 6874 to (226.26, 164.49, 97.46) mm, rotated rx 180 ry 0 rz 180 deg; joints [-145.396, -79.463, -30.733, 63.418, 39.422, -57.068]
  MoveL 6875 to (226.26, 164.49, 97.46) mm, rotated rx 180 ry 0 rz 180 deg; joints [-145.396, -79.463, -30.733, 63.418, 39.422, -57.068]
  Call Extruder(272.61000)
  MoveL 6876 to (225.96, 164.54, 97.46) mm, rotated rx 180 ry 0 rz -180 deg; joints [-145.377, -79.42, -30.82, 63.387, 39.458, -57.018]
  MoveL 6877 to (225.96, 164.54, 97.46) mm, rotated rx 180 ry 0 rz -180 deg; joints [-145.377, -79.42, -30.82, 63.387, 39.458, -57.018]
  Call Extruder(272.76956)
  MoveL 6878 to (225.65, 164.58, 97.46) mm, rotated rx -180 ry 0 rz 180 deg; joints [-145.357, -79.377, -30.907, 63.355, 39.494, -56.969]
  MoveL 6879 to (225.65, 164.58, 97.46) mm, rotated rx -180 ry 0 rz 180 deg; joints [-145.357, -79.377, -30.907, 63.355, 39.494, -56.969]
  Call Extruder(272.92838)
  MoveL 6880 to (225.34, 164.63, 97.46) mm, rotated rx -180 ry 0 rz 180 deg; joints [-145.338, -79.334, -30.994, 63.324, 39.53, -56.92]
  MoveL 6881 to (225.34, 164.63, 97.46) mm, rotated rx -180 ry 0 rz 180 deg; joints [-145.338, -79.334, -30.994, 63.324, 39.53, -56.92]
  Call Extruder(273.10706)
  MoveL 6882 to (225, 164.68, 97.46) mm, rotated rx 180 ry 0 rz 180 deg; joints [-145.317, -79.284, -31.095, 63.287, 39.571, -56.862]
  MoveL 6883 to (225, 164.68, 97.46) mm, rotated rx 180 ry 0 rz 180 deg; joints [-145.317, -79.284, -31.095, 63.287, 39.571, -56.862]
  Call Extruder(273.30550)
  MoveL 6884 to (224.61, 164.72, 97.46) mm, rotated rx 180 ry 0 rz 180 deg; joints [-145.293, -79.229, -31.208, 63.245, 39.616, -56.797]
  MoveL 6885 to (224.61, 164.72, 97.46) mm, rotated rx 180 ry 0 rz 180 deg; joints [-145.293, -79.229, -31.208, 63.245, 39.616, -56.797]
  Call Extruder(273.50307)
  MoveL 6886 to (224.22, 164.77, 97.46) mm, rotated rx -180 ry 0 rz 180 deg; joints [-145.27, -79.173, -31.321, 63.204, 39.662, -56.733]
  MoveL 6887 to (224.22, 164.77, 97.46) mm, rotated rx -180 ry 0 rz 180 deg; joints [-145.27, -79.173, -31.321, 63.204, 39.662, -56.733]
  Call Extruder(273.69978)
  MoveL 6888 to (223.84, 164.82, 97.46) mm, rotated rx 180 ry 0 rz 180 deg; joints [-145.246, -79.118, -31.433, 63.163, 39.707, -56.668]
  MoveL 6889 to (223.84, 164.82, 97.46) mm, rotated rx 180 ry 0 rz 180 deg; joints [-145.246, -79.118, -31.433, 63.163, 39.707, -56.668]
  Call Extruder(273.89562)
  MoveL 6890 to (223.45, 164.86, 97.46) mm, rotated rx 180 ry 0 rz 180 deg; joints [-145.223, -79.062, -31.546, 63.121, 39.752, -56.604]
  MoveL 6891 to (223.45, 164.86, 97.46) mm, rotated rx 180 ry 0 rz 180 deg; joints [-145.223, -79.062, -31.546, 63.121, 39.752, -56.604]
  Call Extruder(274.19098)
  MoveL 6892 to (222.86, 164.91, 97.46) mm, rotated rx 180 ry 0 rz 180 deg; joints [-145.189, -78.976, -31.721, 63.056, 39.821, -56.503]
  MoveL 6893 to (222.86, 164.91, 97.46) mm, rotated rx 180 ry 0 rz 180 deg; joints [-145.189, -78.976, -31.721, 63.056, 39.821, -56.503]
  Call Extruder(274.48500)
  MoveL 6894 to (222.27, 164.95, 97.46) mm, rotated rx 180 ry 0 rz 180 deg; joints [-145.155, -78.89, -31.896, 62.99, 39.89, -56.402]
  MoveL 6895 to (222.27, 164.95, 97.46) mm, rotated rx 180 ry 0 rz 180 deg; joints [-145.155, -78.89, -31.896, 62.99, 39.89, -56.402]
  Call Extruder(274.77770)
  MoveL 6896 to (221.68, 165, 97.46) mm, rotated rx 180 ry 0 rz 180 deg; joints [-145.121, -78.805, -32.069, 62.926, 39.958, -56.302]
  MoveL 6897 to (221.68, 165, 97.46) mm, rotated rx 180 ry 0 rz 180 deg; joints [-145.121, -78.805, -32.069, 62.926, 39.958, -56.302]
  Call Extruder(275.35114)
  MoveL 6898 to (220.52, 165.05, 97.46) mm, rotated rx 180 ry 0 rz 180 deg; joints [-145.056, -78.633, -32.42, 62.792, 40.093, -56.098]
  MoveL 6899 to (220.52, 165.05, 97.46) mm, rotated rx 180 ry 0 rz 180 deg; joints [-145.056, -78.633, -32.42, 62.792, 40.093, -56.098]
  Call Extruder(276.06515)
  MoveL 6900 to (219.06, 165.09, 97.46) mm, rotated rx 180 ry 0 rz -180 deg; joints [-144.977, -78.417, -32.858, 62.626, 40.261, -55.843]
  Call Extruder(392.91189)
  MoveL 6901 to (-19.06, 165.09, 97.46) mm, rotated rx 180 ry 0 rz -180 deg; joints [-127.435, -57.799, -77.724, 61.356, 64.794, -37.942]
  Call Extruder(393.34049)
  MoveL 6902 to (-19.94, 165.07, 97.46) mm, rotated rx 180 ry 0 rz 180 deg; joints [-127.348, -57.754, -77.833, 61.405, 64.878, -37.912]
  MoveL 6903 to (-19.94, 165.07, 97.46) mm, rotated rx 180 ry 0 rz 180 deg; joints [-127.348, -57.754, -77.833, 61.405, 64.878, -37.912]
  Call Extruder(393.91395)
  MoveL 6904 to (-21.1, 165.03, 97.46) mm, rotated rx 180 ry 0 rz 180 deg; joints [-127.235, -57.693, -77.981, 61.468, 64.989, -37.871]
  MoveL 6905 to (-21.1, 165.03, 97.46) mm, rotated rx 180 ry 0 rz 180 deg; joints [-127.235, -57.693, -77.981, 61.468, 64.989, -37.871]
  Call Extruder(394.34824)
  MoveL 6906 to (-21.97, 164.98, 97.46) mm, rotated rx 180 ry 0 rz -180 deg; joints [-127.15, -57.646, -78.094, 61.515, 65.073, -37.838]
  MoveL 6907 to (-21.97, 164.98, 97.46) mm, rotated rx 180 ry 0 rz -180 deg; joints [-127.15, -57.646, -78.094, 61.515, 65.073, -37.838]
  Call Extruder(394.64227)
  MoveL 6908 to (-22.56, 164.93, 97.46) mm, rotated rx 180 ry 0 rz -180 deg; joints [-127.093, -57.614, -78.172, 61.545, 65.129, -37.814]
  MoveL 6909 to (-22.56, 164.93, 97.46) mm, rotated rx 180 ry 0 rz -180 deg; joints [-127.093, -57.614, -78.172, 61.545, 65.129, -37.814]
  Call Extruder(394.93763)
  MoveL 6910 to (-23.15, 164.89, 97.46) mm, rotated rx 180 ry 0 rz 180 deg; joints [-127.037, -57.581, -78.25, 61.576, 65.185, -37.79]
  MoveL 6911 to (-23.15, 164.89, 97.46) mm, rotated rx 180 ry 0 rz 180 deg; joints [-127.037, -57.581, -78.25, 61.576, 65.185, -37.79]
  Call Extruder(395.18385)
  MoveL 6912 to (-23.64, 164.84, 97.46) mm, rotated rx 180 ry 0 rz 180 deg; joints [-126.991, -57.554, -78.316, 61.6, 65.232, -37.77]
  MoveL 6913 to (-23.64, 164.84, 97.46) mm, rotated rx 180 ry 0 rz 180 deg; joints [-126.991, -57.554, -78.316, 61.6, 65.232, -37.77]
  Call Extruder(395.38056)
  MoveL 6914 to (-24.03, 164.79, 97.46) mm, rotated rx -180 ry 0 rz 180 deg; joints [-126.955, -57.532, -78.37, 61.618, 65.269, -37.752]
  MoveL 6915 to (-24.03, 164.79, 97.46) mm, rotated rx -180 ry 0 rz 180 deg; joints [-126.955, -57.532, -78.37, 61.618, 65.269, -37.752]
  Call Extruder(395.57813)
  MoveL 6916 to (-24.42, 164.75, 97.46) mm, rotated rx -180 ry 0 rz 180 deg; joints [-126.919, -57.51, -78.423, 61.637, 65.305, -37.735]
  MoveL 6917 to (-24.42, 164.75, 97.46) mm, rotated rx -180 ry 0 rz 180 deg; joints [-126.919, -57.51, -78.423, 61.637, 65.305, -37.735]
  Call Extruder(395.77657)
  MoveL 6918 to (-24.8, 164.7, 97.46) mm, rotated rx 180 ry 0 rz -180 deg; joints [-126.883, -57.488, -78.477, 61.656, 65.342, -37.718]
  MoveL 6919 to (-24.8, 164.7, 97.46) mm, rotated rx 180 ry 0 rz -180 deg; joints [-126.883, -57.488, -78.477, 61.656, 65.342, -37.718]
  Call Extruder(395.97588)
  MoveL 6920 to (-25.19, 164.66, 97.46) mm, rotated rx 180 ry 0 rz -180 deg; joints [-126.847, -57.466, -78.53, 61.674, 65.379, -37.7]
  MoveL 6921 to (-25.19, 164.66, 97.46) mm, rotated rx 180 ry 0 rz -180 deg; joints [-126.847, -57.466, -78.53, 61.674, 65.379, -37.7]
  Call Extruder(396.13471)
  MoveL 6922 to (-25.5, 164.61, 97.46) mm, rotated rx 180 ry 0 rz 180 deg; joints [-126.82, -57.447, -78.574, 61.688, 65.408, -37.685]
  MoveL 6923 to (-25.5, 164.61, 97.46) mm, rotated rx 180 ry 0 rz 180 deg; joints [-126.82, -57.447, -78.574, 61.688, 65.408, -37.685]
  Call Extruder(396.29427)
  MoveL 6924 to (-25.8, 164.56, 97.46) mm, rotated rx -180 ry 0 rz 180 deg; joints [-126.792, -57.429, -78.618, 61.701, 65.437, -37.67]
  MoveL 6925 to (-25.8, 164.56, 97.46) mm, rotated rx -180 ry 0 rz 180 deg; joints [-126.792, -57.429, -78.618, 61.701, 65.437, -37.67]
  Call Extruder(396.45456)
  MoveL 6926 to (-26.11, 164.51, 97.46) mm, rotated rx 180 ry 0 rz -180 deg; joints [-126.765, -57.411, -78.662, 61.715, 65.466, -37.655]
  MoveL 6927 to (-26.11, 164.51, 97.46) mm, rotated rx 180 ry 0 rz -180 deg; joints [-126.765, -57.411, -78.662, 61.715, 65.466, -37.655]
  Call Extruder(396.61557)
  MoveL 6928 to (-26.41, 164.46, 97.46) mm, rotated rx -180 ry 0 rz -180 deg; joints [-126.737, -57.393, -78.706, 61.729, 65.496, -37.64]
  MoveL 6929 to (-26.41, 164.46, 97.46) mm, rotated rx -180 ry 0 rz -180 deg; joints [-126.737, -57.393, -78.706, 61.729, 65.496, -37.64]
  Call Extruder(396.77732)
  MoveL 6930 to (-26.72, 164.41, 97.46) mm, rotated rx 180 ry 0 rz 180 deg; joints [-126.71, -57.375, -78.75, 61.742, 65.525, -37.625]
  MoveL 6931 to (-26.72, 164.41, 97.46) mm, rotated rx 180 ry 0 rz 180 deg; joints [-126.71, -57.375, -78.75, 61.742, 65.525, -37.625]
  Call Extruder(396.93979)
  MoveL 6932 to (-27.03, 164.36, 97.46) mm, rotated rx -180 ry 0 rz 180 deg; joints [-126.682, -57.357, -78.794, 61.756, 65.554, -37.61]
  MoveL 6933 to (-27.03, 164.36, 97.46) mm, rotated rx -180 ry 0 rz 180 deg; joints [-126.682, -57.357, -78.794, 61.756, 65.554, -37.61]
  Call Extruder(397.07371)
  MoveL 6934 to (-27.27, 164.32, 97.46) mm, rotated rx 180 ry 0 rz 180 deg; joints [-126.66, -57.341, -78.831, 61.766, 65.577, -37.597]
  MoveL 6935 to (-27.27, 164.32, 97.46) mm, rotated rx 180 ry 0 rz 180 deg; joints [-126.66, -57.341, -78.831, 61.766, 65.577, -37.597]
  Call Extruder(397.20825)
  MoveL 6936 to (-27.52, 164.27, 97.46) mm, rotated rx -180 ry 0 rz 180 deg; joints [-126.638, -57.326, -78.868, 61.776, 65.601, -37.583]
  MoveL 6937 to (-27.52, 164.27, 97.46) mm, rotated rx -180 ry 0 rz 180 deg; joints [-126.638, -57.326, -78.868, 61.776, 65.601, -37.583]
  Call Extruder(397.34340)
  MoveL 6938 to (-27.77, 164.22, 97.46) mm, rotated rx 180 ry 0 rz 180 deg; joints [-126.617, -57.311, -78.906, 61.786, 65.625, -37.57]
  MoveL 6939 to (-27.77, 164.22, 97.46) mm, rotated rx 180 ry 0 rz 180 deg; joints [-126.617, -57.311, -78.906, 61.786, 65.625, -37.57]
  Call Extruder(397.47915)
  MoveL 6940 to (-28.02, 164.17, 97.46) mm, rotated rx -180 ry 0 rz 180 deg; joints [-126.595, -57.295, -78.943, 61.797, 65.648, -37.557]
  MoveL 6941 to (-28.02, 164.17, 97.46) mm, rotated rx -180 ry 0 rz 180 deg; joints [-126.595, -57.295, -78.943, 61.797, 65.648, -37.557]
  Call Extruder(397.61552)
  MoveL 6942 to (-28.27, 164.12, 97.46) mm, rotated rx -180 ry 0 rz 180 deg; joints [-126.573, -57.28, -78.98, 61.807, 65.672, -37.543]
  MoveL 6943 to (-28.27, 164.12, 97.46) mm, rotated rx -180 ry 0 rz 180 deg; joints [-126.573, -57.28, -78.98, 61.807, 65.672, -37.543]
  Call Extruder(397.70039)
  MoveL 6944 to (-28.42, 164.09, 97.46) mm, rotated rx -180 ry 0 rz 180 deg; joints [-126.559, -57.27, -79.003, 61.813, 65.687, -37.535]
  Set speed (130.0 mm/s)
  MoveL 6945 to (-31.76, 163.31, 97.46) mm, rotated rx 180 ry 0 rz 180 deg; joints [-126.274, -57.059, -79.517, 61.942, 66.003, -37.344]
  MoveL 6946 to (-31.76, 163.31, 106.87) mm, rotated rx 180 ry 0 rz 180 deg; joints [-126.274, -55.796, -80.061, 62.227, 65.666, -38.041]
  Call Extruder(395.70039)
  Set speed (40.0 mm/s)
  MoveL 6947 to (-31.76, 163.31, 106.87) mm, rotated rx 180 ry 0 rz 180 deg; joints [-126.274, -55.796, -80.061, 62.227, 65.666, -38.041]
  Call Extruder(0.00000)
  Set speed (130.0 mm/s)
  MoveL 6948 to (-31.64, 163.21, 106.87) mm, rotated rx -180 ry 0 rz 180 deg; joints [-126.294, -55.795, -80.063, 62.209, 65.654, -38.032]
  Call Extruder(2.00000)
  Set speed (40.0 mm/s)
  MoveL 6949 to (-31.64, 163.21, 106.87) mm, rotated rx -180 ry 0 rz 180 deg; joints [-126.294, -55.795, -80.063, 62.209, 65.654, -38.032]
  Set speed (30.0 mm/s)
  MoveL 6950 to (-31.64, 163.21, 106.87) mm, rotated rx -180 ry 0 rz 180 deg; joints [-126.294, -55.795, -80.063, 62.209, 65.654, -38.032]
  Call Extruder(2.18198)
  MoveL 6951 to (-31.93, 163.09, 106.87) mm, rotated rx 180 ry 0 rz -180 deg; joints [-126.273, -55.773, -80.116, 62.215, 65.682, -38.01]
  MoveL 6952 to (-31.93, 163.09, 106.87) mm, rotated rx 180 ry 0 rz -180 deg; joints [-126.273, -55.773, -80.116, 62.215, 65.682, -38.01]
  Call Extruder(2.36471)
  MoveL 6953 to (-32.22, 162.96, 106.87) mm, rotated rx 180 ry 0 rz 180 deg; joints [-126.252, -55.751, -80.169, 62.221, 65.709, -37.987]
  MoveL 6954 to (-32.22, 162.96, 106.87) mm, rotated rx 180 ry 0 rz 180 deg; joints [-126.252, -55.751, -80.169, 62.221, 65.709, -37.987]
  Call Extruder(2.53513)
  MoveL 6955 to (-32.49, 162.85, 106.87) mm, rotated rx 180 ry 0 rz 180 deg; joints [-126.233, -55.73, -80.219, 62.226, 65.734, -37.966]
  MoveL 6956 to (-32.49, 162.85, 106.87) mm, rotated rx 180 ry 0 rz 180 deg; joints [-126.233, -55.73, -80.219, 62.226, 65.734, -37.966]
  Call Extruder(2.69310)
  MoveL 6957 to (-32.74, 162.74, 106.87) mm, rotated rx -180 ry 0 rz 180 deg; joints [-126.215, -55.711, -80.265, 62.231, 65.758, -37.947]
  MoveL 6958 to (-32.74, 162.74, 106.87) mm, rotated rx -180 ry 0 rz 180 deg; joints [-126.215, -55.711, -80.265, 62.231, 65.758, -37.947]
  Call Extruder(2.85168)
  MoveL 6959 to (-32.99, 162.64, 106.87) mm, rotated rx 180 ry 0 rz 180 deg; joints [-126.197, -55.692, -80.31, 62.236, 65.781, -37.927]
  MoveL 6960 to (-32.99, 162.64, 106.87) mm, rotated rx 180 ry 0 rz 180 deg; joints [-126.197, -55.692, -80.31, 62.236, 65.781, -37.927]
  Call Extruder(3.05785)
  MoveL 6961 to (-33.29, 162.46, 106.87) mm, rotated rx -180 ry 0 rz 180 deg; joints [-126.179, -55.666, -80.373, 62.237, 65.81, -37.898]
  MoveL 6962 to (-33.29, 162.46, 106.87) mm, rotated rx -180 ry 0 rz 180 deg; joints [-126.179, -55.666, -80.373, 62.237, 65.81, -37.898]
  Call Extruder(3.26479)
  MoveL 6963 to (-33.6, 162.29, 106.87) mm, rotated rx 180 ry 0 rz 180 deg; joints [-126.16, -55.639, -80.436, 62.239, 65.838, -37.869]
  MoveL 6964 to (-33.6, 162.29, 106.87) mm, rotated rx 180 ry 0 rz 180 deg; joints [-126.16, -55.639, -80.436, 62.239, 65.838, -37.869]
  Call Extruder(3.47251)
  MoveL 6965 to (-33.9, 162.11, 106.87) mm, rotated rx 180 ry 0 rz -180 deg; joints [-126.142, -55.613, -80.499, 62.24, 65.866, -37.84]
  MoveL 6966 to (-33.9, 162.11, 106.87) mm, rotated rx 180 ry 0 rz -180 deg; joints [-126.142, -55.613, -80.499, 62.24, 65.866, -37.84]
  Call Extruder(3.68101)
  MoveL 6967 to (-34.21, 161.94, 106.87) mm, rotated rx 180 ry 0 rz 180 deg; joints [-126.123, -55.587, -80.562, 62.241, 65.895, -37.811]
  MoveL 6968 to (-34.21, 161.94, 106.87) mm, rotated rx 180 ry 0 rz 180 deg; joints [-126.123, -55.587, -80.562, 62.241, 65.895, -37.811]
  Call Extruder(3.86055)
  MoveL 6969 to (-34.45, 161.76, 106.87) mm, rotated rx 180 ry 0 rz 180 deg; joints [-126.111, -55.563, -80.618, 62.239, 65.917, -37.784]
  MoveL 6970 to (-34.45, 161.76, 106.87) mm, rotated rx 180 ry 0 rz 180 deg; joints [-126.111, -55.563, -80.618, 62.239, 65.917, -37.784]
  Call Extruder(4.19399)
  MoveL 6971 to (-34.9, 161.43, 106.87) mm, rotated rx 180 ry 0 rz -180 deg; joints [-126.089, -55.52, -80.722, 62.234, 65.959, -37.733]
  MoveL 6972 to (-34.9, 161.43, 106.87) mm, rotated rx 180 ry 0 rz -180 deg; joints [-126.089, -55.52, -80.722, 62.234, 65.959, -37.733]
  Call Extruder(4.52861)
  MoveL 6973 to (-35.35, 161.1, 106.87) mm, rotated rx -180 ry 0 rz 180 deg; joints [-126.067, -55.477, -80.826, 62.23, 66.001, -37.682]
  Call Extruder(5.35652)
  MoveL 6974 to (-36.39, 160.19, 106.87) mm, rotated rx -180 ry 0 rz 180 deg; joints [-126.027, -55.367, -81.089, 62.204, 66.097, -37.547]
  Call Extruder(6.18445)
  MoveL 6975 to (-37.3, 159.15, 106.87) mm, rotated rx -180 ry 0 rz 180 deg; joints [-126.011, -55.256, -81.357, 62.157, 66.18, -37.402]
  Call Extruder(6.35176)
  MoveL 6976 to (-37.47, 158.93, 106.87) mm, rotated rx -180 ry 0 rz -180 deg; joints [-126.011, -55.234, -81.411, 62.144, 66.195, -37.371]
  MoveL 6977 to (-37.47, 158.93, 106.87) mm, rotated rx -180 ry 0 rz -180 deg; joints [-126.011, -55.234, -81.411, 62.144, 66.195, -37.371]
  Call Extruder(6.68519)
  MoveL 6978 to (-37.79, 158.48, 106.87) mm, rotated rx 180 ry 0 rz -180 deg; joints [-126.011, -55.189, -81.519, 62.12, 66.224, -37.31]
  MoveL 6979 to (-37.79, 158.48, 106.87) mm, rotated rx 180 ry 0 rz -180 deg; joints [-126.011, -55.189, -81.519, 62.12, 66.224, -37.31]
  Call Extruder(7.01743)
  MoveL 6980 to (-38.12, 158.03, 106.87) mm, rotated rx 180 ry 0 rz 180 deg; joints [-126.011, -55.144, -81.628, 62.095, 66.254, -37.249]
  MoveL 6981 to (-38.12, 158.03, 106.87) mm, rotated rx 180 ry 0 rz 180 deg; joints [-126.011, -55.144, -81.628, 62.095, 66.254, -37.249]
  Call Extruder(7.13511)
  MoveL 6982 to (-38.22, 157.85, 106.87) mm, rotated rx -180 ry 0 rz 180 deg; joints [-126.013, -55.128, -81.666, 62.084, 66.263, -37.226]
  MoveL 6983 to (-38.22, 157.85, 106.87) mm, rotated rx -180 ry 0 rz 180 deg; joints [-126.013, -55.128, -81.666, 62.084, 66.263, -37.226]
  Call Extruder(7.34283)
  MoveL 6984 to (-38.4, 157.55, 106.87) mm, rotated rx -180 ry 0 rz -180 deg; joints [-126.018, -55.1, -81.733, 62.064, 66.279, -37.186]
  MoveL 6985 to (-38.4, 157.55, 106.87) mm, rotated rx -180 ry 0 rz -180 deg; joints [-126.018, -55.1, -81.733, 62.064, 66.279, -37.186]
  Call Extruder(7.54978)
  MoveL 6986 to (-38.57, 157.25, 106.87) mm, rotated rx -180 ry 0 rz 180 deg; joints [-126.023, -55.072, -81.801, 62.045, 66.294, -37.146]
  MoveL 6987 to (-38.57, 157.25, 106.87) mm, rotated rx -180 ry 0 rz 180 deg; joints [-126.023, -55.072, -81.801, 62.045, 66.294, -37.146]
  Call Extruder(7.75595)
  MoveL 6988 to (-38.75, 156.94, 106.87) mm, rotated rx -180 ry 0 rz 180 deg; joints [-126.028, -55.044, -81.869, 62.025, 66.31, -37.106]
  MoveL 6989 to (-38.75, 156.94, 106.87) mm, rotated rx -180 ry 0 rz 180 deg; joints [-126.028, -55.044, -81.869, 62.025, 66.31, -37.106]
  Call Extruder(7.93763)
  MoveL 6990 to (-38.89, 156.66, 106.87) mm, rotated rx -180 ry 0 rz 180 deg; joints [-126.034, -55.019, -81.928, 62.006, 66.322, -37.07]
  MoveL 6991 to (-38.89, 156.66, 106.87) mm, rotated rx -180 ry 0 rz 180 deg; joints [-126.034, -55.019, -81.928, 62.006, 66.322, -37.07]
  Call Extruder(8.09561)
  MoveL 6992 to (-39, 156.42, 106.87) mm, rotated rx -180 ry 0 rz -180 deg; joints [-126.042, -54.998, -81.979, 61.988, 66.332, -37.039]
  MoveL 6993 to (-39, 156.42, 106.87) mm, rotated rx -180 ry 0 rz -180 deg; joints [-126.042, -54.998, -81.979, 61.988, 66.332, -37.039]
  Call Extruder(8.25300)
  MoveL 6994 to (-39.1, 156.17, 106.87) mm, rotated rx 180 ry 0 rz 180 deg; joints [-126.05, -54.977, -82.03, 61.969, 66.341, -37.007]
  MoveL 6995 to (-39.1, 156.17, 106.87) mm, rotated rx 180 ry 0 rz 180 deg; joints [-126.05, -54.977, -82.03, 61.969, 66.341, -37.007]
  Call Extruder(8.43571)
  MoveL 6996 to (-39.23, 155.88, 106.87) mm, rotated rx 180 ry 0 rz 180 deg; joints [-126.06, -54.953, -82.09, 61.947, 66.351, -36.97]
  MoveL 6997 to (-39.23, 155.88, 106.87) mm, rotated rx 180 ry 0 rz 180 deg; joints [-126.06, -54.953, -82.09, 61.947, 66.351, -36.97]
  Call Extruder(8.61768)
  MoveL 6998 to (-39.35, 155.58, 106.87) mm, rotated rx 180 ry 0 rz -180 deg; joints [-126.07, -54.928, -82.149, 61.925, 66.362, -36.933]
  MoveL 6999 to (-39.35, 155.58, 106.87) mm, rotated rx 180 ry 0 rz -180 deg; joints [-126.07, -54.928, -82.149, 61.925, 66.362, -36.933]
  Call Extruder(8.76501)
  MoveL 7000 to (-39.44, 155.34, 106.87) mm, rotated rx 180 ry 0 rz 180 deg; joints [-126.079, -54.908, -82.197, 61.906, 66.37, -36.903]
  MoveL 7001 to (-39.44, 155.34, 106.87) mm, rotated rx 180 ry 0 rz 180 deg; joints [-126.079, -54.908, -82.197, 61.906, 66.37, -36.903]
  Call Extruder(8.87825)
  MoveL 7002 to (-39.5, 155.15, 106.87) mm, rotated rx 180 ry 0 rz 180 deg; joints [-126.087, -54.893, -82.233, 61.891, 66.375, -36.879]
  MoveL 7003 to (-39.5, 155.15, 106.87) mm, rotated rx 180 ry 0 rz 180 deg; joints [-126.087, -54.893, -82.233, 61.891, 66.375, -36.879]
  Call Extruder(8.99104)
  MoveL 7004 to (-39.56, 154.97, 106.87) mm, rotated rx -180 ry 0 rz 180 deg; joints [-126.095, -54.878, -82.269, 61.876, 66.38, -36.856]
  MoveL 7005 to (-39.56, 154.97, 106.87) mm, rotated rx -180 ry 0 rz 180 deg; joints [-126.095, -54.878, -82.269, 61.876, 66.38, -36.856]
  Call Extruder(9.10338)
  MoveL 7006 to (-39.62, 154.78, 106.87) mm, rotated rx 180 ry 0 rz 180 deg; joints [-126.103, -54.863, -82.306, 61.86, 66.385, -36.833]
  MoveL 7007 to (-39.62, 154.78, 106.87) mm, rotated rx 180 ry 0 rz 180 deg; joints [-126.103, -54.863, -82.306, 61.86, 66.385, -36.833]
  Call Extruder(9.21528)
  MoveL 7008 to (-39.68, 154.59, 106.87) mm, rotated rx 180 ry 0 rz -180 deg; joints [-126.111, -54.849, -82.342, 61.845, 66.39, -36.809]
  MoveL 7009 to (-39.68, 154.59, 106.87) mm, rotated rx 180 ry 0 rz -180 deg; joints [-126.111, -54.849, -82.342, 61.845, 66.39, -36.809]
  Call Extruder(9.33668)
  MoveL 7010 to (-39.75, 154.38, 106.87) mm, rotated rx 180 ry 0 rz 180 deg; joints [-126.12, -54.832, -82.382, 61.828, 66.396, -36.784]
  MoveL 7011 to (-39.75, 154.38, 106.87) mm, rotated rx 180 ry 0 rz 180 deg; joints [-126.12, -54.832, -82.382, 61.828, 66.396, -36.784]
  Call Extruder(9.46748)
  MoveL 7012 to (-39.82, 154.16, 106.87) mm, rotated rx -180 ry 0 rz 180 deg; joints [-126.131, -54.815, -82.424, 61.81, 66.402, -36.756]
  MoveL 7013 to (-39.82, 154.16, 106.87) mm, rotated rx -180 ry 0 rz 180 deg; joints [-126.131, -54.815, -82.424, 61.81, 66.402, -36.756]
  Call Extruder(9.59770)
  MoveL 7014 to (-39.88, 153.94, 106.87) mm, rotated rx 180 ry 0 rz -180 deg; joints [-126.141, -54.797, -82.466, 61.791, 66.407, -36.728]
  MoveL 7015 to (-39.88, 153.94, 106.87) mm, rotated rx 180 ry 0 rz -180 deg; joints [-126.141, -54.797, -82.466, 61.791, 66.407, -36.728]
  Call Extruder(9.72737)
  MoveL 7016 to (-39.95, 153.71, 106.87) mm, rotated rx -180 ry 0 rz 180 deg; joints [-126.151, -54.78, -82.509, 61.772, 66.413, -36.701]
  MoveL 7017 to (-39.95, 153.71, 106.87) mm, rotated rx -180 ry 0 rz 180 deg; joints [-126.151, -54.78, -82.509, 61.772, 66.413, -36.701]
  Call Extruder(9.85647)
  MoveL 7018 to (-40.02, 153.49, 106.87) mm, rotated rx 180 ry 0 rz 180 deg; joints [-126.161, -54.762, -82.551, 61.754, 66.419, -36.673]
  MoveL 7019 to (-40.02, 153.49, 106.87) mm, rotated rx 180 ry 0 rz 180 deg; joints [-126.161, -54.762, -82.551, 61.754, 66.419, -36.673]
  Call Extruder(9.97156)
  MoveL 7020 to (-40.06, 153.28, 106.87) mm, rotated rx 180 ry 0 rz 180 deg; joints [-126.173, -54.747, -82.588, 61.736, 66.422, -36.648]
  MoveL 7021 to (-40.06, 153.28, 106.87) mm, rotated rx 180 ry 0 rz 180 deg; joints [-126.173, -54.747, -82.588, 61.736, 66.422, -36.648]
  Call Extruder(10.08619)
  MoveL 7022 to (-40.11, 153.08, 106.87) mm, rotated rx 180 ry 0 rz 180 deg; joints [-126.184, -54.732, -82.625, 61.718, 66.426, -36.624]
  MoveL 7023 to (-40.11, 153.08, 106.87) mm, rotated rx 180 ry 0 rz 180 deg; joints [-126.184, -54.732, -82.625, 61.718, 66.426, -36.624]
  Call Extruder(10.20037)
  MoveL 7024 to (-40.15, 152.88, 106.87) mm, rotated rx -180 ry 0 rz 180 deg; joints [-126.195, -54.717, -82.662, 61.699, 66.429, -36.599]
  MoveL 7025 to (-40.15, 152.88, 106.87) mm, rotated rx -180 ry 0 rz 180 deg; joints [-126.195, -54.717, -82.662, 61.699, 66.429, -36.599]
  Call Extruder(10.31410)
  MoveL 7026 to (-40.2, 152.67, 106.87) mm, rotated rx -180 ry 0 rz 180 deg; joints [-126.206, -54.702, -82.698, 61.681, 66.433, -36.574]
  MoveL 7027 to (-40.2, 152.67, 106.87) mm, rotated rx -180 ry 0 rz 180 deg; joints [-126.206, -54.702, -82.698, 61.681, 66.433, -36.574]
  Call Extruder(10.43953)
  MoveL 7028 to (-40.24, 152.45, 106.87) mm, rotated rx 180 ry 0 rz 180 deg; joints [-126.219, -54.685, -82.739, 61.661, 66.437, -36.547]
  MoveL 7029 to (-40.24, 152.45, 106.87) mm, rotated rx 180 ry 0 rz 180 deg; joints [-126.219, -54.685, -82.739, 61.661, 66.437, -36.547]
  Call Extruder(10.57651)
  MoveL 7030 to (-40.29, 152.2, 106.87) mm, rotated rx 180 ry 0 rz 180 deg; joints [-126.233, -54.667, -82.783, 61.638, 66.44, -36.517]
  MoveL 7031 to (-40.29, 152.2, 106.87) mm, rotated rx 180 ry 0 rz 180 deg; joints [-126.233, -54.667, -82.783, 61.638, 66.44, -36.517]
  Call Extruder(10.71287)
  MoveL 7032 to (-40.34, 151.95, 106.87) mm, rotated rx 180 ry 0 rz 180 deg; joints [-126.248, -54.649, -82.827, 61.616, 66.444, -36.487]
  MoveL 7033 to (-40.34, 151.95, 106.87) mm, rotated rx 180 ry 0 rz 180 deg; joints [-126.248, -54.649, -82.827, 61.616, 66.444, -36.487]
  Call Extruder(10.84863)
  MoveL 7034 to (-40.39, 151.7, 106.87) mm, rotated rx 180 ry 0 rz 180 deg; joints [-126.262, -54.631, -82.872, 61.593, 66.448, -36.457]
  MoveL 7035 to (-40.39, 151.7, 106.87) mm, rotated rx 180 ry 0 rz 180 deg; joints [-126.262, -54.631, -82.872, 61.593, 66.448, -36.457]
  Call Extruder(10.98377)
  MoveL 7036 to (-40.44, 151.45, 106.87) mm, rotated rx 180 ry 0 rz 180 deg; joints [-126.276, -54.613, -82.916, 61.571, 66.452, -36.427]
  MoveL 7037 to (-40.44, 151.45, 106.87) mm, rotated rx 180 ry 0 rz 180 deg; joints [-126.276, -54.613, -82.916, 61.571, 66.452, -36.427]
  Call Extruder(11.11831)
  MoveL 7038 to (-40.49, 151.2, 106.87) mm, rotated rx 180 ry 0 rz 180 deg; joints [-126.291, -54.595, -82.96, 61.548, 66.456, -36.397]
  MoveL 7039 to (-40.49, 151.2, 106.87) mm, rotated rx 180 ry 0 rz 180 deg; joints [-126.291, -54.595, -82.96, 61.548, 66.456, -36.397]
  Call Extruder(11.25223)
  MoveL 7040 to (-40.54, 150.95, 106.87) mm, rotated rx 180 ry 0 rz -180 deg; joints [-126.305, -54.576, -83.004, 61.526, 66.46, -36.367]
  MoveL 7041 to (-40.54, 150.95, 106.87) mm, rotated rx 180 ry 0 rz -180 deg; joints [-126.305, -54.576, -83.004, 61.526, 66.46, -36.367]
  Call Extruder(11.40009)
  MoveL 7042 to (-40.59, 150.67, 106.87) mm, rotated rx 180 ry 0 rz 180 deg; joints [-126.322, -54.557, -83.052, 61.5, 66.464, -36.334]
  MoveL 7043 to (-40.59, 150.67, 106.87) mm, rotated rx 180 ry 0 rz 180 deg; joints [-126.322, -54.557, -83.052, 61.5, 66.464, -36.334]
  Call Extruder(11.56181)
  MoveL 7044 to (-40.64, 150.37, 106.87) mm, rotated rx 180 ry 0 rz 180 deg; joints [-126.341, -54.535, -83.105, 61.471, 66.467, -36.297]
  MoveL 7045 to (-40.64, 150.37, 106.87) mm, rotated rx 180 ry 0 rz 180 deg; joints [-126.341, -54.535, -83.105, 61.471, 66.467, -36.297]
  Call Extruder(11.72281)
  MoveL 7046 to (-40.69, 150.06, 106.87) mm, rotated rx -180 ry 0 rz 180 deg; joints [-126.36, -54.513, -83.158, 61.443, 66.471, -36.261]
  MoveL 7047 to (-40.69, 150.06, 106.87) mm, rotated rx -180 ry 0 rz 180 deg; joints [-126.36, -54.513, -83.158, 61.443, 66.471, -36.261]
  Call Extruder(11.88308)
  MoveL 7048 to (-40.74, 149.76, 106.87) mm, rotated rx 180 ry 0 rz -180 deg; joints [-126.379, -54.492, -83.21, 61.414, 66.474, -36.224]
  MoveL 7049 to (-40.74, 149.76, 106.87) mm, rotated rx 180 ry 0 rz -180 deg; joints [-126.379, -54.492, -83.21, 61.414, 66.474, -36.224]
  Call Extruder(12.04262)
  MoveL 7050 to (-40.78, 149.45, 106.87) mm, rotated rx 180 ry 0 rz 180 deg; joints [-126.398, -54.47, -83.263, 61.386, 66.478, -36.188]
  MoveL 7051 to (-40.78, 149.45, 106.87) mm, rotated rx 180 ry 0 rz 180 deg; joints [-126.398, -54.47, -83.263, 61.386, 66.478, -36.188]
  Call Extruder(12.20143)
  MoveL 7052 to (-40.83, 149.14, 106.87) mm, rotated rx 180 ry 0 rz 180 deg; joints [-126.417, -54.449, -83.315, 61.357, 66.482, -36.152]
  MoveL 7053 to (-40.83, 149.14, 106.87) mm, rotated rx 180 ry 0 rz 180 deg; joints [-126.417, -54.449, -83.315, 61.357, 66.482, -36.152]
  Call Extruder(12.38010)
  MoveL 7054 to (-40.88, 148.8, 106.87) mm, rotated rx 180 ry 0 rz 180 deg; joints [-126.439, -54.425, -83.374, 61.324, 66.485, -36.111]
  MoveL 7055 to (-40.88, 148.8, 106.87) mm, rotated rx 180 ry 0 rz 180 deg; joints [-126.439, -54.425, -83.374, 61.324, 66.485, -36.111]
  Call Extruder(12.57854)
  MoveL 7056 to (-40.92, 148.41, 106.87) mm, rotated rx 180 ry 0 rz 180 deg; joints [-126.465, -54.398, -83.439, 61.286, 66.488, -36.065]
  MoveL 7057 to (-40.92, 148.41, 106.87) mm, rotated rx 180 ry 0 rz 180 deg; joints [-126.465, -54.398, -83.439, 61.286, 66.488, -36.065]
  Call Extruder(12.77611)
  MoveL 7058 to (-40.97, 148.02, 106.87) mm, rotated rx -180 ry 0 rz -180 deg; joints [-126.491, -54.372, -83.503, 61.249, 66.491, -36.019]
  MoveL 7059 to (-40.97, 148.02, 106.87) mm, rotated rx -180 ry 0 rz -180 deg; joints [-126.491, -54.372, -83.503, 61.249, 66.491, -36.019]
  Call Extruder(12.97282)
  MoveL 7060 to (-41.02, 147.63, 106.87) mm, rotated rx 180 ry 0 rz 180 deg; joints [-126.517, -54.346, -83.568, 61.211, 66.494, -35.973]
  MoveL 7061 to (-41.02, 147.63, 106.87) mm, rotated rx 180 ry 0 rz 180 deg; joints [-126.517, -54.346, -83.568, 61.211, 66.494, -35.973]
  Call Extruder(13.16865)
  MoveL 7062 to (-41.06, 147.25, 106.87) mm, rotated rx -180 ry 0 rz 180 deg; joints [-126.543, -54.319, -83.632, 61.174, 66.497, -35.928]
  MoveL 7063 to (-41.06, 147.25, 106.87) mm, rotated rx -180 ry 0 rz 180 deg; joints [-126.543, -54.319, -83.632, 61.174, 66.497, -35.928]
  Call Extruder(13.46405)
  MoveL 7064 to (-41.11, 146.66, 106.87) mm, rotated rx -180 ry 0 rz 180 deg; joints [-126.585, -54.28, -83.728, 61.115, 66.5, -35.859]
  MoveL 7065 to (-41.11, 146.66, 106.87) mm, rotated rx -180 ry 0 rz 180 deg; joints [-126.585, -54.28, -83.728, 61.115, 66.5, -35.859]
  Call Extruder(13.75812)
  MoveL 7066 to (-41.16, 146.07, 106.87) mm, rotated rx -180 ry 0 rz 180 deg; joints [-126.628, -54.241, -83.823, 61.056, 66.502, -35.79]
  MoveL 7067 to (-41.16, 146.07, 106.87) mm, rotated rx -180 ry 0 rz 180 deg; joints [-126.628, -54.241, -83.823, 61.056, 66.502, -35.79]
  Call Extruder(14.05086)
  MoveL 7068 to (-41.2, 145.48, 106.87) mm, rotated rx 180 ry 0 rz 180 deg; joints [-126.67, -54.203, -83.919, 60.997, 66.505, -35.721]
  MoveL 7069 to (-41.2, 145.48, 106.87) mm, rotated rx 180 ry 0 rz 180 deg; joints [-126.67, -54.203, -83.919, 60.997, 66.505, -35.721]
  Call Extruder(14.62431)
  MoveL 7070 to (-41.25, 144.32, 106.87) mm, rotated rx 180 ry 0 rz -180 deg; joints [-126.759, -54.128, -84.101, 60.877, 66.506, -35.587]
  MoveL 7071 to (-41.25, 144.32, 106.87) mm, rotated rx 180 ry 0 rz -180 deg; joints [-126.759, -54.128, -84.101, 60.877, 66.506, -35.587]
  Call Extruder(15.33827)
  MoveL 7072 to (-41.29, 142.86, 106.87) mm, rotated rx -180 ry 0 rz 180 deg; joints [-126.873, -54.037, -84.326, 60.725, 66.505, -35.419]
  Call Extruder(57.40309)
  MoveL 7073 to (-41.29, 57.14, 106.87) mm, rotated rx 180 ry 0 rz 180 deg; joints [-135.148, -49.543, -96.04, 50.334, 66.378, -25.791]
  Call Extruder(57.83165)
  MoveL 7074 to (-41.27, 56.26, 106.87) mm, rotated rx -180 ry 0 rz 180 deg; joints [-135.25, -49.506, -96.144, 50.212, 66.377, -25.695]
  MoveL 7075 to (-41.27, 56.26, 106.87) mm, rotated rx -180 ry 0 rz 180 deg; joints [-135.25, -49.506, -96.144, 50.212, 66.377, -25.695]
  Call Extruder(58.11773)
  MoveL 7076 to (-41.25, 55.68, 106.87) mm, rotated rx 180 ry 0 rz 180 deg; joints [-135.318, -49.482, -96.211, 50.129, 66.375, -25.631]
  MoveL 7077 to (-41.25, 55.68, 106.87) mm, rotated rx 180 ry 0 rz 180 deg; joints [-135.318, -49.482, -96.211, 50.129, 66.375, -25.631]
  Call Extruder(58.69247)
  MoveL 7078 to (-41.2, 54.52, 106.87) mm, rotated rx 180 ry 0 rz 180 deg; joints [-135.457, -49.434, -96.346, 49.964, 66.371, -25.504]
  MoveL 7079 to (-41.2, 54.52, 106.87) mm, rotated rx 180 ry 0 rz 180 deg; joints [-135.457, -49.434, -96.346, 49.964, 66.371, -25.504]
  Call Extruder(58.98587)
  MoveL 7080 to (-41.16, 53.93, 106.87) mm, rotated rx -180 ry 0 rz -180 deg; joints [-135.53, -49.41, -96.412, 49.878, 66.367, -25.44]
  MoveL 7081 to (-41.16, 53.93, 106.87) mm, rotated rx -180 ry 0 rz -180 deg; joints [-135.53, -49.41, -96.412, 49.878, 66.367, -25.44]
  Call Extruder(59.28060)
  MoveL 7082 to (-41.11, 53.34, 106.87) mm, rotated rx -180 ry 0 rz -180 deg; joints [-135.603, -49.387, -96.477, 49.792, 66.362, -25.376]
  MoveL 7083 to (-41.11, 53.34, 106.87) mm, rotated rx -180 ry 0 rz -180 deg; joints [-135.603, -49.387, -96.477, 49.792, 66.362, -25.376]
  Call Extruder(59.57666)
  MoveL 7084 to (-41.06, 52.75, 106.87) mm, rotated rx 180 ry 0 rz 180 deg; joints [-135.676, -49.364, -96.542, 49.705, 66.358, -25.312]
  MoveL 7085 to (-41.06, 52.75, 106.87) mm, rotated rx 180 ry 0 rz 180 deg; joints [-135.676, -49.364, -96.542, 49.705, 66.358, -25.312]
  Call Extruder(59.77293)
  MoveL 7086 to (-41.02, 52.37, 106.87) mm, rotated rx 180 ry 0 rz 180 deg; joints [-135.726, -49.349, -96.583, 49.647, 66.354, -25.27]
  MoveL 7087 to (-41.02, 52.37, 106.87) mm, rotated rx 180 ry 0 rz 180 deg; joints [-135.726, -49.349, -96.583, 49.647, 66.354, -25.27]
  Call Extruder(59.97007)
  MoveL 7088 to (-40.97, 51.98, 106.87) mm, rotated rx 180 ry 0 rz 180 deg; joints [-135.776, -49.335, -96.624, 49.589, 66.349, -25.228]
  MoveL 7089 to (-40.97, 51.98, 106.87) mm, rotated rx 180 ry 0 rz 180 deg; joints [-135.776, -49.335, -96.624, 49.589, 66.349, -25.228]
  Call Extruder(60.16808)
  MoveL 7090 to (-40.92, 51.59, 106.87) mm, rotated rx 180 ry 0 rz -180 deg; joints [-135.827, -49.32, -96.665, 49.531, 66.345, -25.187]
  MoveL 7091 to (-40.92, 51.59, 106.87) mm, rotated rx 180 ry 0 rz -180 deg; joints [-135.827, -49.32, -96.665, 49.531, 66.345, -25.187]
  Call Extruder(60.36695)
  MoveL 7092 to (-40.88, 51.2, 106.87) mm, rotated rx 180 ry 0 rz 180 deg; joints [-135.877, -49.306, -96.706, 49.472, 66.341, -25.145]
  MoveL 7093 to (-40.88, 51.2, 106.87) mm, rotated rx 180 ry 0 rz 180 deg; joints [-135.877, -49.306, -96.706, 49.472, 66.341, -25.145]
  Call Extruder(60.54603)
  MoveL 7094 to (-40.83, 50.86, 106.87) mm, rotated rx 180 ry 0 rz 180 deg; joints [-135.922, -49.293, -96.741, 49.419, 66.336, -25.108]
  MoveL 7095 to (-40.83, 50.86, 106.87) mm, rotated rx 180 ry 0 rz 180 deg; joints [-135.922, -49.293, -96.741, 49.419, 66.336, -25.108]
  Call Extruder(60.70521)
  MoveL 7096 to (-40.78, 50.55, 106.87) mm, rotated rx -180 ry 0 rz 180 deg; joints [-135.964, -49.283, -96.772, 49.372, 66.332, -25.075]
  MoveL 7097 to (-40.78, 50.55, 106.87) mm, rotated rx -180 ry 0 rz 180 deg; joints [-135.964, -49.283, -96.772, 49.372, 66.332, -25.075]
  Call Extruder(60.86512)
  MoveL 7098 to (-40.73, 50.24, 106.87) mm, rotated rx 180 ry 0 rz -180 deg; joints [-136.005, -49.272, -96.802, 49.325, 66.327, -25.042]
  MoveL 7099 to (-40.73, 50.24, 106.87) mm, rotated rx 180 ry 0 rz -180 deg; joints [-136.005, -49.272, -96.802, 49.325, 66.327, -25.042]
  Call Extruder(61.02575)
  MoveL 7100 to (-40.69, 49.94, 106.87) mm, rotated rx 180 ry 0 rz -180 deg; joints [-136.046, -49.261, -96.832, 49.278, 66.323, -25.01]
  MoveL 7101 to (-40.69, 49.94, 106.87) mm, rotated rx 180 ry 0 rz -180 deg; joints [-136.046, -49.261, -96.832, 49.278, 66.323, -25.01]
  Call Extruder(61.18711)
  MoveL 7102 to (-40.64, 49.63, 106.87) mm, rotated rx 180 ry 0 rz 180 deg; joints [-136.087, -49.25, -96.863, 49.23, 66.318, -24.977]
  MoveL 7103 to (-40.64, 49.63, 106.87) mm, rotated rx 180 ry 0 rz 180 deg; joints [-136.087, -49.25, -96.863, 49.23, 66.318, -24.977]
  Call Extruder(61.34920)
  MoveL 7104 to (-40.59, 49.33, 106.87) mm, rotated rx 180 ry 0 rz -180 deg; joints [-136.128, -49.24, -96.893, 49.183, 66.313, -24.945]
  MoveL 7105 to (-40.59, 49.33, 106.87) mm, rotated rx 180 ry 0 rz -180 deg; joints [-136.128, -49.24, -96.893, 49.183, 66.313, -24.945]
  Call Extruder(61.49740)
  MoveL 7106 to (-40.54, 49.05, 106.87) mm, rotated rx 180 ry 0 rz -180 deg; joints [-136.166, -49.23, -96.92, 49.139, 66.309, -24.915]
  MoveL 7107 to (-40.54, 49.05, 106.87) mm, rotated rx 180 ry 0 rz -180 deg; joints [-136.166, -49.23, -96.92, 49.139, 66.309, -24.915]
  Call Extruder(61.63163)
  MoveL 7108 to (-40.49, 48.8, 106.87) mm, rotated rx -180 ry 0 rz -180 deg; joints [-136.201, -49.222, -96.944, 49.1, 66.304, -24.889]
  MoveL 7109 to (-40.49, 48.8, 106.87) mm, rotated rx -180 ry 0 rz -180 deg; joints [-136.201, -49.222, -96.944, 49.1, 66.304, -24.889]
  Call Extruder(61.76647)
  MoveL 7110 to (-40.44, 48.55, 106.87) mm, rotated rx 180 ry 0 rz -180 deg; joints [-136.236, -49.214, -96.967, 49.06, 66.299, -24.862]
  MoveL 7111 to (-40.44, 48.55, 106.87) mm, rotated rx 180 ry 0 rz -180 deg; joints [-136.236, -49.214, -96.967, 49.06, 66.299, -24.862]
  Call Extruder(61.90192)
  MoveL 7112 to (-40.39, 48.3, 106.87) mm, rotated rx 180 ry 0 rz 180 deg; joints [-136.271, -49.205, -96.99, 49.021, 66.295, -24.836]
  MoveL 7113 to (-40.39, 48.3, 106.87) mm, rotated rx 180 ry 0 rz 180 deg; joints [-136.271, -49.205, -96.99, 49.021, 66.295, -24.836]
  Call Extruder(62.03798)
  MoveL 7114 to (-40.34, 48.05, 106.87) mm, rotated rx 180 ry 0 rz 180 deg; joints [-136.306, -49.197, -97.014, 48.981, 66.29, -24.81]
  MoveL 7115 to (-40.34, 48.05, 106.87) mm, rotated rx 180 ry 0 rz 180 deg; joints [-136.306, -49.197, -97.014, 48.981, 66.29, -24.81]
  Call Extruder(62.17465)
  MoveL 7116 to (-40.29, 47.8, 106.87) mm, rotated rx 180 ry 0 rz 180 deg; joints [-136.341, -49.189, -97.037, 48.941, 66.285, -24.783]
  MoveL 7117 to (-40.29, 47.8, 106.87) mm, rotated rx 180 ry 0 rz 180 deg; joints [-136.341, -49.189, -97.037, 48.941, 66.285, -24.783]
  Call Extruder(62.31193)
  MoveL 7118 to (-40.24, 47.55, 106.87) mm, rotated rx 180 ry 0 rz 180 deg; joints [-136.376, -49.181, -97.06, 48.902, 66.28, -24.757]
  MoveL 7119 to (-40.24, 47.55, 106.87) mm, rotated rx 180 ry 0 rz 180 deg; joints [-136.376, -49.181, -97.06, 48.902, 66.28, -24.757]
  Call Extruder(62.43760)
  MoveL 7120 to (-40.2, 47.33, 106.87) mm, rotated rx 180 ry 0 rz 180 deg; joints [-136.408, -49.173, -97.081, 48.866, 66.276, -24.733]
  MoveL 7121 to (-40.2, 47.33, 106.87) mm, rotated rx 180 ry 0 rz 180 deg; joints [-136.408, -49.173, -97.081, 48.866, 66.276, -24.733]
  Call Extruder(62.55156)
  MoveL 7122 to (-40.15, 47.12, 106.87) mm, rotated rx 180 ry 0 rz 180 deg; joints [-136.437, -49.167, -97.1, 48.833, 66.272, -24.711]
  MoveL 7123 to (-40.15, 47.12, 106.87) mm, rotated rx 180 ry 0 rz 180 deg; joints [-136.437, -49.167, -97.1, 48.833, 66.272, -24.711]
  Call Extruder(62.66597)
  MoveL 7124 to (-40.11, 46.92, 106.87) mm, rotated rx 180 ry 0 rz 180 deg; joints [-136.466, -49.16, -97.118, 48.8, 66.267, -24.69]
  MoveL 7125 to (-40.11, 46.92, 106.87) mm, rotated rx 180 ry 0 rz 180 deg; joints [-136.466, -49.16, -97.118, 48.8, 66.267, -24.69]
  Call Extruder(62.78083)
  MoveL 7126 to (-40.06, 46.72, 106.87) mm, rotated rx 180 ry 0 rz 180 deg; joints [-136.495, -49.154, -97.137, 48.767, 66.263, -24.668]
  MoveL 7127 to (-40.06, 46.72, 106.87) mm, rotated rx 180 ry 0 rz 180 deg; joints [-136.495, -49.154, -97.137, 48.767, 66.263, -24.668]
  Call Extruder(62.89614)
  MoveL 7128 to (-40.02, 46.51, 106.87) mm, rotated rx 180 ry 0 rz 180 deg; joints [-136.525, -49.147, -97.155, 48.734, 66.259, -24.647]
  MoveL 7129 to (-40.02, 46.51, 106.87) mm, rotated rx 180 ry 0 rz 180 deg; joints [-136.525, -49.147, -97.155, 48.734, 66.259, -24.647]
  Call Extruder(63.02552)
  MoveL 7130 to (-39.95, 46.29, 106.87) mm, rotated rx 180 ry 0 rz 180 deg; joints [-136.559, -49.141, -97.173, 48.696, 66.252, -24.624]
  MoveL 7131 to (-39.95, 46.29, 106.87) mm, rotated rx 180 ry 0 rz 180 deg; joints [-136.559, -49.141, -97.173, 48.696, 66.252, -24.624]
  Call Extruder(63.15547)
  MoveL 7132 to (-39.88, 46.06, 106.87) mm, rotated rx 180 ry 0 rz -180 deg; joints [-136.593, -49.135, -97.191, 48.658, 66.246, -24.6]
  MoveL 7133 to (-39.88, 46.06, 106.87) mm, rotated rx 180 ry 0 rz -180 deg; joints [-136.593, -49.135, -97.191, 48.658, 66.246, -24.6]
  Call Extruder(63.28598)
  MoveL 7134 to (-39.81, 45.84, 106.87) mm, rotated rx -180 ry 0 rz 180 deg; joints [-136.627, -49.128, -97.209, 48.621, 66.239, -24.577]
  MoveL 7135 to (-39.81, 45.84, 106.87) mm, rotated rx -180 ry 0 rz 180 deg; joints [-136.627, -49.128, -97.209, 48.621, 66.239, -24.577]
  Call Extruder(63.41705)
  MoveL 7136 to (-39.75, 45.62, 106.87) mm, rotated rx 180 ry 0 rz 180 deg; joints [-136.661, -49.122, -97.227, 48.583, 66.233, -24.554]
  MoveL 7137 to (-39.75, 45.62, 106.87) mm, rotated rx 180 ry 0 rz 180 deg; joints [-136.661, -49.122, -97.227, 48.583, 66.233, -24.554]
  Call Extruder(63.53870)
  MoveL 7138 to (-39.68, 45.41, 106.87) mm, rotated rx -180 ry 0 rz 180 deg; joints [-136.693, -49.116, -97.243, 48.548, 66.226, -24.533]
  MoveL 7139 to (-39.68, 45.41, 106.87) mm, rotated rx -180 ry 0 rz 180 deg; joints [-136.693, -49.116, -97.243, 48.548, 66.226, -24.533]
  Call Extruder(63.65082)
  MoveL 7140 to (-39.62, 45.22, 106.87) mm, rotated rx 180 ry 0 rz 180 deg; joints [-136.722, -49.111, -97.258, 48.516, 66.22, -24.513]
  MoveL 7141 to (-39.62, 45.22, 106.87) mm, rotated rx 180 ry 0 rz 180 deg; joints [-136.722, -49.111, -97.258, 48.516, 66.22, -24.513]
  Call Extruder(63.76339)
  MoveL 7142 to (-39.56, 45.03, 106.87) mm, rotated rx 180 ry 0 rz 180 deg; joints [-136.751, -49.106, -97.272, 48.483, 66.214, -24.494]
  MoveL 7143 to (-39.56, 45.03, 106.87) mm, rotated rx 180 ry 0 rz 180 deg; joints [-136.751, -49.106, -97.272, 48.483, 66.214, -24.494]
  Call Extruder(63.87640)
  MoveL 7144 to (-39.5, 44.85, 106.87) mm, rotated rx 180 ry 0 rz -180 deg; joints [-136.781, -49.101, -97.287, 48.451, 66.209, -24.474]
  MoveL 7145 to (-39.5, 44.85, 106.87) mm, rotated rx 180 ry 0 rz -180 deg; joints [-136.781, -49.101, -97.287, 48.451, 66.209, -24.474]
  Call Extruder(63.98986)
  MoveL 7146 to (-39.44, 44.66, 106.87) mm, rotated rx 180 ry 0 rz -180 deg; joints [-136.81, -49.096, -97.301, 48.419, 66.203, -24.455]
  MoveL 7147 to (-39.44, 44.66, 106.87) mm, rotated rx 180 ry 0 rz -180 deg; joints [-136.81, -49.096, -97.301, 48.419, 66.203, -24.455]
  Call Extruder(64.13750)
  MoveL 7148 to (-39.35, 44.42, 106.87) mm, rotated rx -180 ry 0 rz 180 deg; joints [-136.849, -49.09, -97.318, 48.377, 66.194, -24.431]
  MoveL 7149 to (-39.35, 44.42, 106.87) mm, rotated rx -180 ry 0 rz 180 deg; joints [-136.849, -49.09, -97.318, 48.377, 66.194, -24.431]
  Call Extruder(64.31984)
  MoveL 7150 to (-39.22, 44.13, 106.87) mm, rotated rx 180 ry 0 rz 180 deg; joints [-136.898, -49.083, -97.337, 48.324, 66.182, -24.401]
  MoveL 7151 to (-39.22, 44.13, 106.87) mm, rotated rx 180 ry 0 rz 180 deg; joints [-136.898, -49.083, -97.337, 48.324, 66.182, -24.401]
  Call Extruder(64.50294)
  MoveL 7152 to (-39.11, 43.83, 106.87) mm, rotated rx 180 ry 0 rz 180 deg; joints [-136.946, -49.077, -97.356, 48.272, 66.17, -24.371]
  MoveL 7153 to (-39.11, 43.83, 106.87) mm, rotated rx 180 ry 0 rz 180 deg; joints [-136.946, -49.077, -97.356, 48.272, 66.17, -24.371]
  Call Extruder(64.66062)
  MoveL 7154 to (-39, 43.58, 106.87) mm, rotated rx 180 ry 0 rz -180 deg; joints [-136.988, -49.071, -97.371, 48.227, 66.16, -24.346]
  MoveL 7155 to (-39, 43.58, 106.87) mm, rotated rx 180 ry 0 rz -180 deg; joints [-136.988, -49.071, -97.371, 48.227, 66.16, -24.346]
  Call Extruder(64.81891)
  MoveL 7156 to (-38.89, 43.34, 106.87) mm, rotated rx 180 ry 0 rz 180 deg; joints [-137.029, -49.066, -97.387, 48.182, 66.149, -24.321]
  MoveL 7157 to (-38.89, 43.34, 106.87) mm, rotated rx 180 ry 0 rz 180 deg; joints [-137.029, -49.066, -97.387, 48.182, 66.149, -24.321]
  Call Extruder(65.00093)
  MoveL 7158 to (-38.75, 43.06, 106.87) mm, rotated rx 180 ry 0 rz -180 deg; joints [-137.078, -49.061, -97.402, 48.13, 66.135, -24.294]
  MoveL 7159 to (-38.75, 43.06, 106.87) mm, rotated rx 180 ry 0 rz -180 deg; joints [-137.078, -49.061, -97.402, 48.13, 66.135, -24.294]
  Call Extruder(65.20748)
  MoveL 7160 to (-38.57, 42.75, 106.87) mm, rotated rx -180 ry 0 rz -180 deg; joints [-137.135, -49.056, -97.415, 48.071, 66.118, -24.264]
  MoveL 7161 to (-38.57, 42.75, 106.87) mm, rotated rx -180 ry 0 rz -180 deg; joints [-137.135, -49.056, -97.415, 48.071, 66.118, -24.264]
  Call Extruder(65.41482)
  MoveL 7162 to (-38.4, 42.45, 106.87) mm, rotated rx 180 ry 0 rz -180 deg; joints [-137.191, -49.051, -97.428, 48.012, 66.101, -24.234]
  MoveL 7163 to (-38.4, 42.45, 106.87) mm, rotated rx 180 ry 0 rz -180 deg; joints [-137.191, -49.051, -97.428, 48.012, 66.101, -24.234]
  Call Extruder(65.62293)
  MoveL 7164 to (-38.22, 42.15, 106.87) mm, rotated rx -180 ry 0 rz 180 deg; joints [-137.247, -49.047, -97.442, 47.954, 66.084, -24.205]
  MoveL 7165 to (-38.22, 42.15, 106.87) mm, rotated rx -180 ry 0 rz 180 deg; joints [-137.247, -49.047, -97.442, 47.954, 66.084, -24.205]
  Call Extruder(65.74065)
  MoveL 7166 to (-38.12, 41.98, 106.87) mm, rotated rx 180 ry 0 rz 180 deg; joints [-137.279, -49.044, -97.449, 47.92, 66.074, -24.188]
  MoveL 7167 to (-38.12, 41.98, 106.87) mm, rotated rx 180 ry 0 rz 180 deg; joints [-137.279, -49.044, -97.449, 47.92, 66.074, -24.188]
  Call Extruder(66.07349)
  MoveL 7168 to (-37.8, 41.52, 106.87) mm, rotated rx 180 ry 0 rz 180 deg; joints [-137.37, -49.04, -97.46, 47.827, 66.041, -24.145]
  MoveL 7169 to (-37.8, 41.52, 106.87) mm, rotated rx 180 ry 0 rz 180 deg; joints [-137.37, -49.04, -97.46, 47.827, 66.041, -24.145]
  Call Extruder(66.40752)
  MoveL 7170 to (-37.47, 41.07, 106.87) mm, rotated rx -180 ry 0 rz 180 deg; joints [-137.461, -49.036, -97.471, 47.734, 66.009, -24.103]
  MoveL 7171 to (-37.47, 41.07, 106.87) mm, rotated rx -180 ry 0 rz 180 deg; joints [-137.461, -49.036, -97.471, 47.734, 66.009, -24.103]
  Call Extruder(66.57511)
  MoveL 7172 to (-37.3, 40.85, 106.87) mm, rotated rx 180 ry 0 rz -180 deg; joints [-137.506, -49.035, -97.476, 47.687, 65.993, -24.081]
  Call Extruder(67.40442)
  MoveL 7173 to (-36.39, 39.81, 106.87) mm, rotated rx 180 ry 0 rz -180 deg; joints [-137.733, -49.033, -97.481, 47.46, 65.902, -23.986]
  Call Extruder(68.03549)
  MoveL 7174 to (-35.6, 39.11, 106.87) mm, rotated rx 180 ry 0 rz 180 deg; joints [-137.904, -49.04, -97.461, 47.292, 65.824, -23.926]
  MoveL 7175 to (-35.6, 39.11, 106.87) mm, rotated rx 180 ry 0 rz 180 deg; joints [-137.904, -49.04, -97.461, 47.292, 65.824, -23.926]
  Call Extruder(68.23306)
  MoveL 7176 to (-35.35, 38.9, 106.87) mm, rotated rx 180 ry 0 rz -180 deg; joints [-137.958, -49.042, -97.454, 47.24, 65.799, -23.908]
  Call Extruder(68.56708)
  MoveL 7177 to (-34.9, 38.57, 106.87) mm, rotated rx 180 ry 0 rz 180 deg; joints [-138.048, -49.049, -97.434, 47.154, 65.754, -23.882]
  MoveL 7178 to (-34.9, 38.57, 106.87) mm, rotated rx 180 ry 0 rz 180 deg; joints [-138.048, -49.049, -97.434, 47.154, 65.754, -23.882]
  Call Extruder(68.89991)
  MoveL 7179 to (-34.45, 38.24, 106.87) mm, rotated rx 180 ry 0 rz 180 deg; joints [-138.137, -49.056, -97.414, 47.069, 65.709, -23.855]
  MoveL 7180 to (-34.45, 38.24, 106.87) mm, rotated rx 180 ry 0 rz 180 deg; joints [-138.137, -49.056, -97.414, 47.069, 65.709, -23.855]
  Call Extruder(69.07916)
  MoveL 7181 to (-34.21, 38.07, 106.87) mm, rotated rx 180 ry 0 rz 180 deg; joints [-138.185, -49.06, -97.403, 47.023, 65.685, -23.841]
  MoveL 7182 to (-34.21, 38.07, 106.87) mm, rotated rx 180 ry 0 rz 180 deg; joints [-138.185, -49.06, -97.403, 47.023, 65.685, -23.841]
  Call Extruder(69.28727)
  MoveL 7183 to (-33.9, 37.89, 106.87) mm, rotated rx 180 ry 0 rz -180 deg; joints [-138.24, -49.067, -97.384, 46.972, 65.654, -23.828]
  MoveL 7184 to (-33.9, 37.89, 106.87) mm, rotated rx 180 ry 0 rz -180 deg; joints [-138.24, -49.067, -97.384, 46.972, 65.654, -23.828]
  Call Extruder(69.49460)
  MoveL 7185 to (-33.6, 37.71, 106.87) mm, rotated rx 180 ry 0 rz 180 deg; joints [-138.295, -49.073, -97.365, 46.921, 65.624, -23.815]
  MoveL 7186 to (-33.6, 37.71, 106.87) mm, rotated rx 180 ry 0 rz 180 deg; joints [-138.295, -49.073, -97.365, 46.921, 65.624, -23.815]
  Call Extruder(69.70115)
  MoveL 7187 to (-33.29, 37.54, 106.87) mm, rotated rx 180 ry 0 rz 180 deg; joints [-138.349, -49.08, -97.347, 46.87, 65.593, -23.803]
  MoveL 7188 to (-33.29, 37.54, 106.87) mm, rotated rx 180 ry 0 rz 180 deg; joints [-138.349, -49.08, -97.347, 46.87, 65.593, -23.803]
  Call Extruder(69.90692)
  MoveL 7189 to (-32.99, 37.36, 106.87) mm, rotated rx 180 ry 0 rz 180 deg; joints [-138.404, -49.087, -97.328, 46.819, 65.563, -23.79]
  MoveL 7190 to (-32.99, 37.36, 106.87) mm, rotated rx 180 ry 0 rz 180 deg; joints [-138.404, -49.087, -97.328, 46.819, 65.563, -23.79]
  Call Extruder(70.06523)
  MoveL 7191 to (-32.74, 37.26, 106.87) mm, rotated rx 180 ry 0 rz 180 deg; joints [-138.444, -49.094, -97.308, 46.783, 65.538, -23.783]
  MoveL 7192 to (-32.74, 37.26, 106.87) mm, rotated rx 180 ry 0 rz 180 deg; joints [-138.444, -49.094, -97.308, 46.783, 65.538, -23.783]
  Call Extruder(70.22293)
  MoveL 7193 to (-32.49, 37.15, 106.87) mm, rotated rx 180 ry 0 rz 180 deg; joints [-138.484, -49.101, -97.288, 46.747, 65.513, -23.777]
  MoveL 7194 to (-32.49, 37.15, 106.87) mm, rotated rx 180 ry 0 rz 180 deg; joints [-138.484, -49.101, -97.288, 46.747, 65.513, -23.777]
  Call Extruder(70.39301)
  MoveL 7195 to (-32.22, 37.03, 106.87) mm, rotated rx 180 ry 0 rz 180 deg; joints [-138.527, -49.108, -97.266, 46.708, 65.486, -23.77]
  MoveL 7196 to (-32.22, 37.03, 106.87) mm, rotated rx 180 ry 0 rz 180 deg; joints [-138.527, -49.108, -97.266, 46.708, 65.486, -23.77]
  Call Extruder(70.57535)
  MoveL 7197 to (-31.93, 36.91, 106.87) mm, rotated rx 180 ry 0 rz -180 deg; joints [-138.574, -49.116, -97.243, 46.667, 65.457, -23.763]
  MoveL 7198 to (-31.93, 36.91, 106.87) mm, rotated rx 180 ry 0 rz -180 deg; joints [-138.574, -49.116, -97.243, 46.667, 65.457, -23.763]
  Call Extruder(70.75692)
  MoveL 7199 to (-31.64, 36.79, 106.87) mm, rotated rx 180 ry 0 rz 180 deg; joints [-138.62, -49.125, -97.219, 46.625, 65.427, -23.756]
  MoveL 7200 to (-31.64, 36.79, 106.87) mm, rotated rx 180 ry 0 rz 180 deg; joints [-138.62, -49.125, -97.219, 46.625, 65.427, -23.756]
  Call Extruder(70.87038)
  MoveL 7201 to (-31.45, 36.73, 106.87) mm, rotated rx -180 ry 0 rz 180 deg; joints [-138.648, -49.131, -97.202, 46.601, 65.408, -23.753]
  MoveL 7202 to (-31.45, 36.73, 106.87) mm, rotated rx -180 ry 0 rz 180 deg; joints [-138.648, -49.131, -97.202, 46.601, 65.408, -23.753]
  Call Extruder(70.98339)
  MoveL 7203 to (-31.26, 36.67, 106.87) mm, rotated rx 180 ry 0 rz -180 deg; joints [-138.676, -49.137, -97.184, 46.577, 65.389, -23.751]
  MoveL 7204 to (-31.26, 36.67, 106.87) mm, rotated rx 180 ry 0 rz -180 deg; joints [-138.676, -49.137, -97.184, 46.577, 65.389, -23.751]
  Call Extruder(71.09596)
  MoveL 7205 to (-31.07, 36.61, 106.87) mm, rotated rx -180 ry 0 rz -180 deg; joints [-138.704, -49.143, -97.167, 46.552, 65.371, -23.748]
  MoveL 7206 to (-31.07, 36.61, 106.87) mm, rotated rx -180 ry 0 rz -180 deg; joints [-138.704, -49.143, -97.167, 46.552, 65.371, -23.748]
  Call Extruder(71.20809)
  MoveL 7207 to (-30.88, 36.55, 106.87) mm, rotated rx 180 ry 0 rz 180 deg; joints [-138.732, -49.149, -97.15, 46.528, 65.352, -23.745]
  MoveL 7208 to (-30.88, 36.55, 106.87) mm, rotated rx 180 ry 0 rz 180 deg; joints [-138.732, -49.149, -97.15, 46.528, 65.352, -23.745]
  Call Extruder(71.31977)
  MoveL 7209 to (-30.69, 36.49, 106.87) mm, rotated rx 180 ry 0 rz 180 deg; joints [-138.759, -49.155, -97.132, 46.504, 65.333, -23.742]
  MoveL 7210 to (-30.69, 36.49, 106.87) mm, rotated rx 180 ry 0 rz 180 deg; joints [-138.759, -49.155, -97.132, 46.504, 65.333, -23.742]
  Call Extruder(71.45084)
  MoveL 7211 to (-30.47, 36.42, 106.87) mm, rotated rx 180 ry 0 rz 180 deg; joints [-138.792, -49.163, -97.111, 46.476, 65.31, -23.74]
  MoveL 7212 to (-30.47, 36.42, 106.87) mm, rotated rx 180 ry 0 rz 180 deg; joints [-138.792, -49.163, -97.111, 46.476, 65.31, -23.74]
  Call Extruder(71.58135)
  MoveL 7213 to (-30.25, 36.35, 106.87) mm, rotated rx 180 ry 0 rz -180 deg; joints [-138.824, -49.17, -97.09, 46.448, 65.288, -23.737]
  MoveL 7214 to (-30.25, 36.35, 106.87) mm, rotated rx 180 ry 0 rz -180 deg; joints [-138.824, -49.17, -97.09, 46.448, 65.288, -23.737]
  Call Extruder(71.71129)
  MoveL 7215 to (-30.02, 36.28, 106.87) mm, rotated rx 180 ry 0 rz -180 deg; joints [-138.856, -49.178, -97.069, 46.42, 65.265, -23.734]
  MoveL 7216 to (-30.02, 36.28, 106.87) mm, rotated rx 180 ry 0 rz -180 deg; joints [-138.856, -49.178, -97.069, 46.42, 65.265, -23.734]
  Call Extruder(71.84067)
  MoveL 7217 to (-29.8, 36.22, 106.87) mm, rotated rx 180 ry 0 rz -180 deg; joints [-138.889, -49.185, -97.048, 46.392, 65.243, -23.732]
  MoveL 7218 to (-29.8, 36.22, 106.87) mm, rotated rx 180 ry 0 rz -180 deg; joints [-138.889, -49.185, -97.048, 46.392, 65.243, -23.732]
  Call Extruder(71.96263)
  MoveL 7219 to (-29.59, 36.16, 106.87) mm, rotated rx 180 ry 0 rz -180 deg; joints [-138.919, -49.193, -97.026, 46.366, 65.221, -23.73]
  MoveL 7220 to (-29.59, 36.16, 106.87) mm, rotated rx 180 ry 0 rz -180 deg; joints [-138.919, -49.193, -97.026, 46.366, 65.221, -23.73]
  Call Extruder(72.07748)
  MoveL 7221 to (-29.38, 36.12, 106.87) mm, rotated rx -180 ry 0 rz 180 deg; joints [-138.946, -49.2, -97.005, 46.343, 65.201, -23.73]
  MoveL 7222 to (-29.38, 36.12, 106.87) mm, rotated rx -180 ry 0 rz 180 deg; joints [-138.946, -49.2, -97.005, 46.343, 65.201, -23.73]
  Call Extruder(72.19188)
  MoveL 7223 to (-29.18, 36.07, 106.87) mm, rotated rx -180 ry 0 rz 180 deg; joints [-138.973, -49.208, -96.984, 46.32, 65.18, -23.729]
  MoveL 7224 to (-29.18, 36.07, 106.87) mm, rotated rx -180 ry 0 rz 180 deg; joints [-138.973, -49.208, -96.984, 46.32, 65.18, -23.729]
  Call Extruder(72.30582)
  MoveL 7225 to (-28.97, 36.03, 106.87) mm, rotated rx 180 ry 0 rz -180 deg; joints [-139, -49.215, -96.962, 46.298, 65.16, -23.728]
  MoveL 7226 to (-28.97, 36.03, 106.87) mm, rotated rx 180 ry 0 rz -180 deg; joints [-139, -49.215, -96.962, 46.298, 65.16, -23.728]
  Call Extruder(72.41931)
  MoveL 7227 to (-28.77, 35.98, 106.87) mm, rotated rx -180 ry 0 rz 180 deg; joints [-139.028, -49.223, -96.941, 46.275, 65.139, -23.728]
  MoveL 7228 to (-28.77, 35.98, 106.87) mm, rotated rx -180 ry 0 rz 180 deg; joints [-139.028, -49.223, -96.941, 46.275, 65.139, -23.728]
  Call Extruder(72.55659)
  MoveL 7229 to (-28.52, 35.93, 106.87) mm, rotated rx 180 ry 0 rz -180 deg; joints [-139.06, -49.232, -96.914, 46.247, 65.114, -23.728]
  MoveL 7230 to (-28.52, 35.93, 106.87) mm, rotated rx 180 ry 0 rz -180 deg; joints [-139.06, -49.232, -96.914, 46.247, 65.114, -23.728]
  Call Extruder(72.69326)
  MoveL 7231 to (-28.27, 35.88, 106.87) mm, rotated rx 180 ry 0 rz 180 deg; joints [-139.093, -49.242, -96.887, 46.22, 65.089, -23.728]
  MoveL 7232 to (-28.27, 35.88, 106.87) mm, rotated rx 180 ry 0 rz 180 deg; joints [-139.093, -49.242, -96.887, 46.22, 65.089, -23.728]
  Call Extruder(72.82933)
  MoveL 7233 to (-28.02, 35.83, 106.87) mm, rotated rx 180 ry 0 rz 180 deg; joints [-139.126, -49.251, -96.861, 46.193, 65.064, -23.728]
  MoveL 7234 to (-28.02, 35.83, 106.87) mm, rotated rx 180 ry 0 rz 180 deg; joints [-139.126, -49.251, -96.861, 46.193, 65.064, -23.728]
  Call Extruder(72.96478)
  MoveL 7235 to (-27.77, 35.78, 106.87) mm, rotated rx 180 ry 0 rz 180 deg; joints [-139.158, -49.261, -96.834, 46.166, 65.039, -23.728]
  MoveL 7236 to (-27.77, 35.78, 106.87) mm, rotated rx 180 ry 0 rz 180 deg; joints [-139.158, -49.261, -96.834, 46.166, 65.039, -23.728]
  Call Extruder(73.09962)
  MoveL 7237 to (-27.52, 35.73, 106.87) mm, rotated rx -180 ry 0 rz 180 deg; joints [-139.191, -49.27, -96.807, 46.139, 65.014, -23.727]
  MoveL 7238 to (-27.52, 35.73, 106.87) mm, rotated rx -180 ry 0 rz 180 deg; joints [-139.191, -49.27, -96.807, 46.139, 65.014, -23.727]
  Call Extruder(73.23385)
  MoveL 7239 to (-27.28, 35.68, 106.87) mm, rotated rx 180 ry 0 rz 180 deg; joints [-139.223, -49.279, -96.78, 46.112, 64.989, -23.727]
  MoveL 7240 to (-27.28, 35.68, 106.87) mm, rotated rx 180 ry 0 rz 180 deg; joints [-139.223, -49.279, -96.78, 46.112, 64.989, -23.727]
  Call Extruder(73.36747)
  MoveL 7241 to (-27.03, 35.63, 106.87) mm, rotated rx 180 ry 0 rz 180 deg; joints [-139.256, -49.289, -96.753, 46.085, 64.964, -23.727]
  MoveL 7242 to (-27.03, 35.63, 106.87) mm, rotated rx 180 ry 0 rz 180 deg; joints [-139.256, -49.289, -96.753, 46.085, 64.964, -23.727]
  Call Extruder(73.52957)
  MoveL 7243 to (-26.72, 35.59, 106.87) mm, rotated rx 180 ry 0 rz 180 deg; joints [-139.294, -49.301, -96.719, 46.054, 64.933, -23.729]
  MoveL 7244 to (-26.72, 35.59, 106.87) mm, rotated rx 180 ry 0 rz 180 deg; joints [-139.294, -49.301, -96.719, 46.054, 64.933, -23.729]
  Call Extruder(73.69094)
  MoveL 7245 to (-26.41, 35.54, 106.87) mm, rotated rx -180 ry 0 rz 180 deg; joints [-139.332, -49.313, -96.685, 46.023, 64.902, -23.73]
  MoveL 7246 to (-26.41, 35.54, 106.87) mm, rotated rx -180 ry 0 rz 180 deg; joints [-139.332, -49.313, -96.685, 46.023, 64.902, -23.73]
  Call Extruder(73.85158)
  MoveL 7247 to (-26.11, 35.49, 106.87) mm, rotated rx 180 ry 0 rz -180 deg; joints [-139.371, -49.326, -96.65, 45.992, 64.871, -23.731]
  MoveL 7248 to (-26.11, 35.49, 106.87) mm, rotated rx 180 ry 0 rz -180 deg; joints [-139.371, -49.326, -96.65, 45.992, 64.871, -23.731]
  Call Extruder(74.01150)
  MoveL 7249 to (-25.8, 35.44, 106.87) mm, rotated rx 180 ry 0 rz 180 deg; joints [-139.409, -49.338, -96.616, 45.961, 64.84, -23.732]
  MoveL 7250 to (-25.8, 35.44, 106.87) mm, rotated rx 180 ry 0 rz 180 deg; joints [-139.409, -49.338, -96.616, 45.961, 64.84, -23.732]
  Call Extruder(74.17069)
  MoveL 7251 to (-25.5, 35.39, 106.87) mm, rotated rx -180 ry 0 rz 180 deg; joints [-139.447, -49.35, -96.581, 45.929, 64.809, -23.734]
  MoveL 7252 to (-25.5, 35.39, 106.87) mm, rotated rx -180 ry 0 rz 180 deg; joints [-139.447, -49.35, -96.581, 45.929, 64.809, -23.734]
  Call Extruder(74.32915)
  MoveL 7253 to (-25.19, 35.34, 106.87) mm, rotated rx 180 ry 0 rz 180 deg; joints [-139.485, -49.362, -96.547, 45.898, 64.779, -23.735]
  MoveL 7254 to (-25.19, 35.34, 106.87) mm, rotated rx 180 ry 0 rz 180 deg; joints [-139.485, -49.362, -96.547, 45.898, 64.779, -23.735]
  Call Extruder(74.52802)
  MoveL 7255 to (-24.8, 35.3, 106.87) mm, rotated rx -180 ry 0 rz -180 deg; joints [-139.531, -49.378, -96.501, 45.862, 64.74, -23.738]
  MoveL 7256 to (-24.8, 35.3, 106.87) mm, rotated rx -180 ry 0 rz -180 deg; joints [-139.531, -49.378, -96.501, 45.862, 64.74, -23.738]
  Call Extruder(74.72603)
  MoveL 7257 to (-24.42, 35.25, 106.87) mm, rotated rx 180 ry 0 rz 180 deg; joints [-139.577, -49.395, -96.456, 45.825, 64.7, -23.742]
  MoveL 7258 to (-24.42, 35.25, 106.87) mm, rotated rx 180 ry 0 rz 180 deg; joints [-139.577, -49.395, -96.456, 45.825, 64.7, -23.742]
  Call Extruder(74.92317)
  MoveL 7259 to (-24.03, 35.21, 106.87) mm, rotated rx 180 ry 0 rz 180 deg; joints [-139.624, -49.411, -96.41, 45.788, 64.661, -23.745]
  MoveL 7260 to (-24.03, 35.21, 106.87) mm, rotated rx 180 ry 0 rz 180 deg; joints [-139.624, -49.411, -96.41, 45.788, 64.661, -23.745]
  Call Extruder(75.11944)
  MoveL 7261 to (-23.64, 35.16, 106.87) mm, rotated rx 180 ry 0 rz 180 deg; joints [-139.67, -49.427, -96.364, 45.751, 64.622, -23.748]
  MoveL 7262 to (-23.64, 35.16, 106.87) mm, rotated rx 180 ry 0 rz 180 deg; joints [-139.67, -49.427, -96.364, 45.751, 64.622, -23.748]
  Call Extruder(75.36513)
  MoveL 7263 to (-23.15, 35.11, 106.87) mm, rotated rx 180 ry 0 rz -180 deg; joints [-139.726, -49.448, -96.305, 45.707, 64.573, -23.754]
  MoveL 7264 to (-23.15, 35.11, 106.87) mm, rotated rx 180 ry 0 rz -180 deg; joints [-139.726, -49.448, -96.305, 45.707, 64.573, -23.754]
  Call Extruder(75.65986)
  MoveL 7265 to (-22.56, 35.07, 106.87) mm, rotated rx 180 ry 0 rz -180 deg; joints [-139.793, -49.474, -96.233, 45.655, 64.513, -23.761]
  MoveL 7266 to (-22.56, 35.07, 106.87) mm, rotated rx 180 ry 0 rz -180 deg; joints [-139.793, -49.474, -96.233, 45.655, 64.513, -23.761]
  Call Extruder(75.95326)
  MoveL 7267 to (-21.97, 35.02, 106.87) mm, rotated rx -180 ry 0 rz 180 deg; joints [-139.86, -49.5, -96.161, 45.603, 64.454, -23.769]
  MoveL 7268 to (-21.97, 35.02, 106.87) mm, rotated rx -180 ry 0 rz 180 deg; joints [-139.86, -49.5, -96.161, 45.603, 64.454, -23.769]
  Call Extruder(76.38658)
  MoveL 7269 to (-21.1, 34.98, 106.87) mm, rotated rx 180 ry 0 rz 180 deg; joints [-139.956, -49.539, -96.05, 45.53, 64.365, -23.783]
  MoveL 7270 to (-21.1, 34.98, 106.87) mm, rotated rx 180 ry 0 rz 180 deg; joints [-139.956, -49.539, -96.05, 45.53, 64.365, -23.783]
  Call Extruder(76.95875)
  MoveL 7271 to (-19.94, 34.93, 106.87) mm, rotated rx 180 ry 0 rz 180 deg; joints [-140.081, -49.593, -95.901, 45.435, 64.248, -23.804]
  MoveL 7272 to (-19.94, 34.93, 106.87) mm, rotated rx 180 ry 0 rz 180 deg; joints [-140.081, -49.593, -95.901, 45.435, 64.248, -23.804]
  Call Extruder(77.38658)
  MoveL 7273 to (-19.06, 34.91, 106.87) mm, rotated rx 180 ry 0 rz 180 deg; joints [-140.173, -49.633, -95.787, 45.367, 64.16, -23.821]
  Call Extruder(194.03526)
  MoveL 7274 to (219.06, 34.91, 106.87) mm, rotated rx -180 ry 0 rz 180 deg; joints [-155.896, -67.718, -53.434, 40.856, 38.631, -34.044]
  MoveL 7275 to (219.06, 34.91, 106.87) mm, rotated rx -180 ry 0 rz 180 deg; joints [-155.896, -67.718, -53.434, 40.856, 38.631, -34.044]
  Call Extruder(194.75084)
  MoveL 7276 to (220.52, 34.95, 106.87) mm, rotated rx -180 ry 0 rz 180 deg; joints [-155.953, -67.885, -53.077, 40.935, 38.456, -34.183]
  MoveL 7277 to (220.52, 34.95, 106.87) mm, rotated rx -180 ry 0 rz 180 deg; joints [-155.953, -67.885, -53.077, 40.935, 38.456, -34.183]
  Call Extruder(195.32557)
  MoveL 7278 to (221.68, 35, 106.87) mm, rotated rx 180 ry 0 rz -180 deg; joints [-155.997, -68.021, -52.79, 41.003, 38.317, -34.298]
  MoveL 7279 to (221.68, 35, 106.87) mm, rotated rx 180 ry 0 rz -180 deg; joints [-155.997, -68.021, -52.79, 41.003, 38.317, -34.298]
  Call Extruder(195.61897)
  MoveL 7280 to (222.27, 35.05, 106.87) mm, rotated rx 180 ry 0 rz 180 deg; joints [-156.017, -68.091, -52.641, 41.042, 38.246, -34.361]
  MoveL 7281 to (222.27, 35.05, 106.87) mm, rotated rx 180 ry 0 rz 180 deg; joints [-156.017, -68.091, -52.641, 41.042, 38.246, -34.361]
  Call Extruder(195.91369)
  MoveL 7282 to (222.86, 35.09, 106.87) mm, rotated rx 180 ry 0 rz -180 deg; joints [-156.037, -68.161, -52.492, 41.081, 38.176, -34.423]
  MoveL 7283 to (222.86, 35.09, 106.87) mm, rotated rx 180 ry 0 rz -180 deg; joints [-156.037, -68.161, -52.492, 41.081, 38.176, -34.423]
  Call Extruder(196.20975)
  MoveL 7284 to (223.45, 35.14, 106.87) mm, rotated rx 180 ry 0 rz 180 deg; joints [-156.057, -68.232, -52.343, 41.12, 38.105, -34.486]
  MoveL 7285 to (223.45, 35.14, 106.87) mm, rotated rx 180 ry 0 rz 180 deg; joints [-156.057, -68.232, -52.343, 41.12, 38.105, -34.486]
  Call Extruder(196.40602)
  MoveL 7286 to (223.83, 35.18, 106.87) mm, rotated rx 180 ry 0 rz 180 deg; joints [-156.068, -68.279, -52.243, 41.149, 38.059, -34.53]
  MoveL 7287 to (223.83, 35.18, 106.87) mm, rotated rx 180 ry 0 rz 180 deg; joints [-156.068, -68.279, -52.243, 41.149, 38.059, -34.53]
  Call Extruder(196.60317)
  MoveL 7288 to (224.22, 35.23, 106.87) mm, rotated rx -180 ry 0 rz -180 deg; joints [-156.08, -68.326, -52.142, 41.178, 38.012, -34.575]
  MoveL 7289 to (224.22, 35.23, 106.87) mm, rotated rx -180 ry 0 rz -180 deg; joints [-156.08, -68.326, -52.142, 41.178, 38.012, -34.575]
  Call Extruder(196.80118)
  MoveL 7290 to (224.61, 35.27, 106.87) mm, rotated rx 180 ry 0 rz 180 deg; joints [-156.092, -68.374, -52.042, 41.207, 37.966, -34.619]
  MoveL 7291 to (224.61, 35.27, 106.87) mm, rotated rx 180 ry 0 rz 180 deg; joints [-156.092, -68.374, -52.042, 41.207, 37.966, -34.619]
  Call Extruder(197.00005)
  MoveL 7292 to (225, 35.32, 106.87) mm, rotated rx 180 ry 0 rz -180 deg; joints [-156.103, -68.421, -51.941, 41.236, 37.919, -34.664]
  MoveL 7293 to (225, 35.32, 106.87) mm, rotated rx 180 ry 0 rz -180 deg; joints [-156.103, -68.421, -51.941, 41.236, 37.919, -34.664]
  Call Extruder(197.17913)
  MoveL 7294 to (225.34, 35.37, 106.87) mm, rotated rx 180 ry 0 rz 180 deg; joints [-156.113, -68.464, -51.851, 41.264, 37.878, -34.705]
  MoveL 7295 to (225.34, 35.37, 106.87) mm, rotated rx 180 ry 0 rz 180 deg; joints [-156.113, -68.464, -51.851, 41.264, 37.878, -34.705]
  Call Extruder(197.33831)
  MoveL 7296 to (225.65, 35.42, 106.87) mm, rotated rx 180 ry 0 rz 180 deg; joints [-156.121, -68.502, -51.77, 41.289, 37.841, -34.742]
  MoveL 7297 to (225.65, 35.42, 106.87) mm, rotated rx 180 ry 0 rz 180 deg; joints [-156.121, -68.502, -51.77, 41.289, 37.841, -34.742]
  Call Extruder(197.49823)
  MoveL 7298 to (225.96, 35.47, 106.87) mm, rotated rx 180 ry 0 rz 180 deg; joints [-156.129, -68.54, -51.689, 41.315, 37.804, -34.78]
  MoveL 7299 to (225.96, 35.47, 106.87) mm, rotated rx 180 ry 0 rz 180 deg; joints [-156.129, -68.54, -51.689, 41.315, 37.804, -34.78]
  Call Extruder(197.65886)
  MoveL 7300 to (226.26, 35.51, 106.87) mm, rotated rx 180 ry 0 rz 180 deg; joints [-156.137, -68.579, -51.608, 41.341, 37.768, -34.817]
  MoveL 7301 to (226.26, 35.51, 106.87) mm, rotated rx 180 ry 0 rz 180 deg; joints [-156.137, -68.579, -51.608, 41.341, 37.768, -34.817]
  Call Extruder(197.82023)
  MoveL 7302 to (226.57, 35.56, 106.87) mm, rotated rx 180 ry 0 rz 180 deg; joints [-156.145, -68.617, -51.527, 41.366, 37.731, -34.855]
  MoveL 7303 to (226.57, 35.56, 106.87) mm, rotated rx 180 ry 0 rz 180 deg; joints [-156.145, -68.617, -51.527, 41.366, 37.731, -34.855]
  Call Extruder(197.98233)
  MoveL 7304 to (226.87, 35.61, 106.87) mm, rotated rx 180 ry 0 rz 180 deg; joints [-156.153, -68.656, -51.445, 41.392, 37.695, -34.893]
  MoveL 7305 to (226.87, 35.61, 106.87) mm, rotated rx 180 ry 0 rz 180 deg; joints [-156.153, -68.656, -51.445, 41.392, 37.695, -34.893]
  Call Extruder(198.13052)
  MoveL 7306 to (227.15, 35.66, 106.87) mm, rotated rx 180 ry 0 rz 180 deg; joints [-156.16, -68.691, -51.371, 41.417, 37.661, -34.928]
  MoveL 7307 to (227.15, 35.66, 106.87) mm, rotated rx 180 ry 0 rz 180 deg; joints [-156.16, -68.691, -51.371, 41.417, 37.661, -34.928]
  Call Extruder(198.26476)
  MoveL 7308 to (227.4, 35.71, 106.87) mm, rotated rx 180 ry 0 rz 180 deg; joints [-156.165, -68.723, -51.304, 41.44, 37.631, -34.96]
  MoveL 7309 to (227.4, 35.71, 106.87) mm, rotated rx 180 ry 0 rz 180 deg; joints [-156.165, -68.723, -51.304, 41.44, 37.631, -34.96]
  Call Extruder(198.39960)
  MoveL 7310 to (227.65, 35.76, 106.87) mm, rotated rx -180 ry 0 rz 180 deg; joints [-156.171, -68.755, -51.236, 41.463, 37.602, -34.993]
  MoveL 7311 to (227.65, 35.76, 106.87) mm, rotated rx -180 ry 0 rz 180 deg; joints [-156.171, -68.755, -51.236, 41.463, 37.602, -34.993]
  Call Extruder(198.53505)
  MoveL 7312 to (227.9, 35.81, 106.87) mm, rotated rx 180 ry 0 rz 180 deg; joints [-156.176, -68.787, -51.169, 41.486, 37.572, -35.026]
  MoveL 7313 to (227.9, 35.81, 106.87) mm, rotated rx 180 ry 0 rz 180 deg; joints [-156.176, -68.787, -51.169, 41.486, 37.572, -35.026]
  Call Extruder(198.67111)
  MoveL 7314 to (228.15, 35.86, 106.87) mm, rotated rx 180 ry 0 rz 180 deg; joints [-156.182, -68.819, -51.101, 41.509, 37.542, -35.059]
  MoveL 7315 to (228.15, 35.86, 106.87) mm, rotated rx 180 ry 0 rz 180 deg; joints [-156.182, -68.819, -51.101, 41.509, 37.542, -35.059]
  Call Extruder(198.80779)
  MoveL 7316 to (228.4, 35.91, 106.87) mm, rotated rx 180 ry 0 rz 180 deg; joints [-156.187, -68.851, -51.033, 41.533, 37.512, -35.092]
  MoveL 7317 to (228.4, 35.91, 106.87) mm, rotated rx 180 ry 0 rz 180 deg; joints [-156.187, -68.851, -51.033, 41.533, 37.512, -35.092]
  Call Extruder(198.94507)
  MoveL 7318 to (228.65, 35.96, 106.87) mm, rotated rx 180 ry 0 rz -180 deg; joints [-156.193, -68.883, -50.966, 41.556, 37.482, -35.125]
  MoveL 7319 to (228.65, 35.96, 106.87) mm, rotated rx 180 ry 0 rz -180 deg; joints [-156.193, -68.883, -50.966, 41.556, 37.482, -35.125]
  Call Extruder(199.07074)
  MoveL 7320 to (228.87, 36, 106.87) mm, rotated rx 180 ry 0 rz 180 deg; joints [-156.198, -68.912, -50.904, 41.578, 37.455, -35.155]
  MoveL 7321 to (228.87, 36, 106.87) mm, rotated rx 180 ry 0 rz 180 deg; joints [-156.198, -68.912, -50.904, 41.578, 37.455, -35.155]
  Call Extruder(199.18469)
  MoveL 7322 to (229.08, 36.05, 106.87) mm, rotated rx -180 ry 0 rz 180 deg; joints [-156.202, -68.939, -50.847, 41.598, 37.43, -35.183]
  MoveL 7323 to (229.08, 36.05, 106.87) mm, rotated rx -180 ry 0 rz 180 deg; joints [-156.202, -68.939, -50.847, 41.598, 37.43, -35.183]
  Call Extruder(199.29909)
